// TIA Portal V17 export
// export: Created 2023-04-26T11:43:36.2466218Z, ExportSetting None, DisplayName Totally Integrated Automation Portal, DisplayVersion V17 Update 4, DisplayName TIA Portal Openness, DisplayVersion V17 Update 4, DisplayName TIA Portal Version Control Interface, DisplayVersion V17, DisplayName STEP 7 Professional, DisplayVersion V17 Update 4, DisplayName STEP 7 Safety, DisplayVersion V17, DisplayName WinCC Advanced / Unified PC, DisplayVersion V17 Update 4
FUNCTION "FC_AIn" : Void   // FC14, LAD
TITLE = FC_AIn
{ S7_Optimized_Access := 'FALSE' }
// Analog Input
// stored: SetENOAutomatically false
BEGIN

REGION Network 1: AI 1
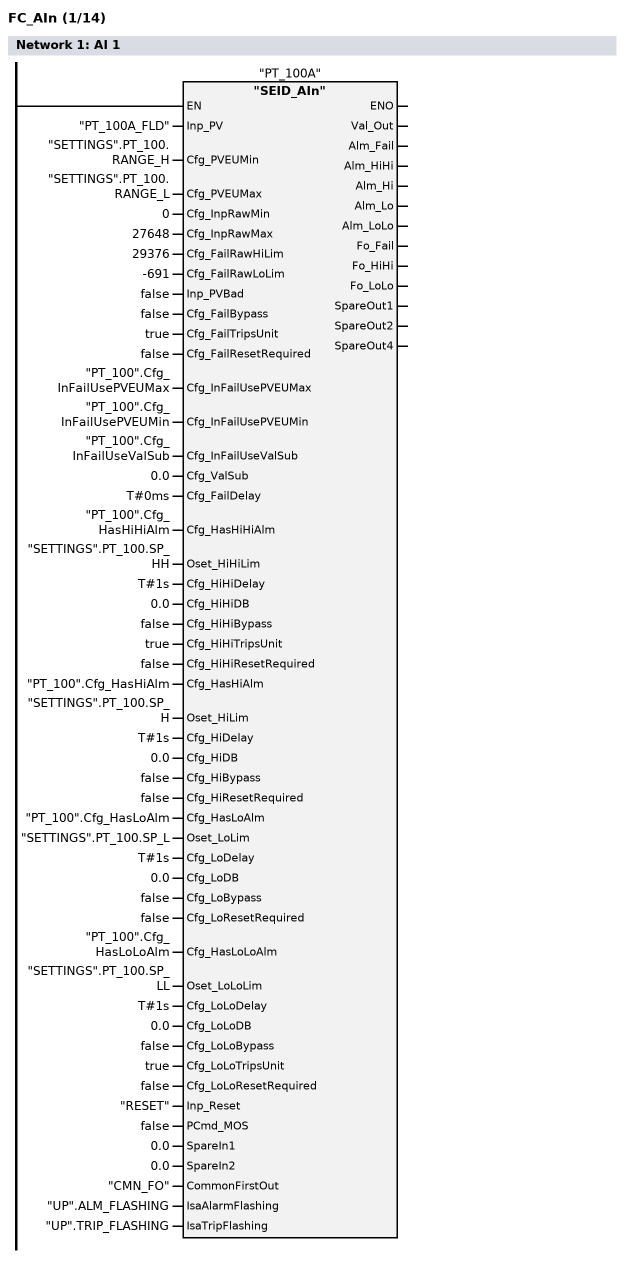
   RUNG wire#powerrail
      "PT_100A"(Inp_PV := "PT_100A_FLD", Cfg_PVEUMin := "SETTINGS".PT_100.RANGE_H, Cfg_PVEUMax := "SETTINGS".PT_100.RANGE_L, Cfg_InpRawMin := 0, Cfg_InpRawMax := 27648, Cfg_FailRawHiLim := 29376, Cfg_FailRawLoLim := -691, Inp_PVBad := false, Cfg_FailBypass := false, Cfg_FailTripsUnit := true, Cfg_FailResetRequired := false, Cfg_InFailUsePVEUMax := "PT_100".Cfg_InFailUsePVEUMax, Cfg_InFailUsePVEUMin := "PT_100".Cfg_InFailUsePVEUMin, Cfg_InFailUseValSub := "PT_100".Cfg_InFailUseValSub, Cfg_ValSub := 0.0, Cfg_FailDelay := T#0ms, Cfg_HasHiHiAlm := "PT_100".Cfg_HasHiHiAlm, Oset_HiHiLim := "SETTINGS".PT_100.SP_HH, Cfg_HiHiDelay := T#1s, Cfg_HiHiDB := 0.0, Cfg_HiHiBypass := false, Cfg_HiHiTripsUnit := true, Cfg_HiHiResetRequired := false, Cfg_HasHiAlm := "PT_100".Cfg_HasHiAlm, Oset_HiLim := "SETTINGS".PT_100.SP_H, Cfg_HiDelay := T#1s, Cfg_HiDB := 0.0, Cfg_HiBypass := false, Cfg_HiResetRequired := false, Cfg_HasLoAlm := "PT_100".Cfg_HasLoAlm, Oset_LoLim := "SETTINGS".PT_100.SP_L, Cfg_LoDelay := T#1s, Cfg_LoDB := 0.0, Cfg_LoBypass := false, Cfg_LoResetRequired := false, Cfg_HasLoLoAlm := "PT_100".Cfg_HasLoLoAlm, Oset_LoLoLim := "SETTINGS".PT_100.SP_LL, Cfg_LoLoDelay := T#1s, Cfg_LoLoDB := 0.0, Cfg_LoLoBypass := false, Cfg_LoLoTripsUnit := true, Cfg_LoLoResetRequired := false, Inp_Reset := "RESET", PCmd_MOS := false, SpareIn1 := 0.0, SpareIn2 := 0.0, CommonFirstOut := "CMN_FO", IsaAlarmFlashing := "UP".ALM_FLASHING, IsaTripFlashing := "UP".TRIP_FLASHING, Val_Out =>, Alm_Fail =>, Alm_HiHi =>, Alm_Hi =>, Alm_Lo =>, Alm_LoLo =>, Fo_Fail =>, Fo_HiHi =>, Fo_LoLo =>, SpareOut1 =>, SpareOut2 =>, SpareOut4 =>)
   END_RUNG
   // the same network as SCL:
   "PT_100A"(Inp_PV := "PT_100A_FLD",   // "SEID_AIn"
             Cfg_PVEUMin := "SETTINGS".PT_100.RANGE_H,
             Cfg_PVEUMax := "SETTINGS".PT_100.RANGE_L,
             Cfg_InpRawMin := 0,
             Cfg_InpRawMax := 27648,
             Cfg_FailRawHiLim := 29376,
             Cfg_FailRawLoLim := -691,
             Inp_PVBad := false,
             Cfg_FailBypass := false,
             Cfg_FailTripsUnit := true,
             Cfg_FailResetRequired := false,
             Cfg_InFailUsePVEUMax := "PT_100".Cfg_InFailUsePVEUMax,
             Cfg_InFailUsePVEUMin := "PT_100".Cfg_InFailUsePVEUMin,
             Cfg_InFailUseValSub := "PT_100".Cfg_InFailUseValSub,
             Cfg_ValSub := 0.0,
             Cfg_FailDelay := T#0ms,
             Cfg_HasHiHiAlm := "PT_100".Cfg_HasHiHiAlm,
             Oset_HiHiLim := "SETTINGS".PT_100.SP_HH,
             Cfg_HiHiDelay := T#1s,
             Cfg_HiHiDB := 0.0,
             Cfg_HiHiBypass := false,
             Cfg_HiHiTripsUnit := true,
             Cfg_HiHiResetRequired := false,
             Cfg_HasHiAlm := "PT_100".Cfg_HasHiAlm,
             Oset_HiLim := "SETTINGS".PT_100.SP_H,
             Cfg_HiDelay := T#1s,
             Cfg_HiDB := 0.0,
             Cfg_HiBypass := false,
             Cfg_HiResetRequired := false,
             Cfg_HasLoAlm := "PT_100".Cfg_HasLoAlm,
             Oset_LoLim := "SETTINGS".PT_100.SP_L,
             Cfg_LoDelay := T#1s,
             Cfg_LoDB := 0.0,
             Cfg_LoBypass := false,
             Cfg_LoResetRequired := false,
             Cfg_HasLoLoAlm := "PT_100".Cfg_HasLoLoAlm,
             Oset_LoLoLim := "SETTINGS".PT_100.SP_LL,
             Cfg_LoLoDelay := T#1s,
             Cfg_LoLoDB := 0.0,
             Cfg_LoLoBypass := false,
             Cfg_LoLoTripsUnit := true,
             Cfg_LoLoResetRequired := false,
             Inp_Reset := "RESET",
             PCmd_MOS := false,
             SpareIn1 := 0.0,
             SpareIn2 := 0.0,
             CommonFirstOut := "CMN_FO",
             IsaAlarmFlashing := "UP".ALM_FLASHING,
             IsaTripFlashing := "UP".TRIP_FLASHING);
END_REGION

REGION Network 2: AI 2
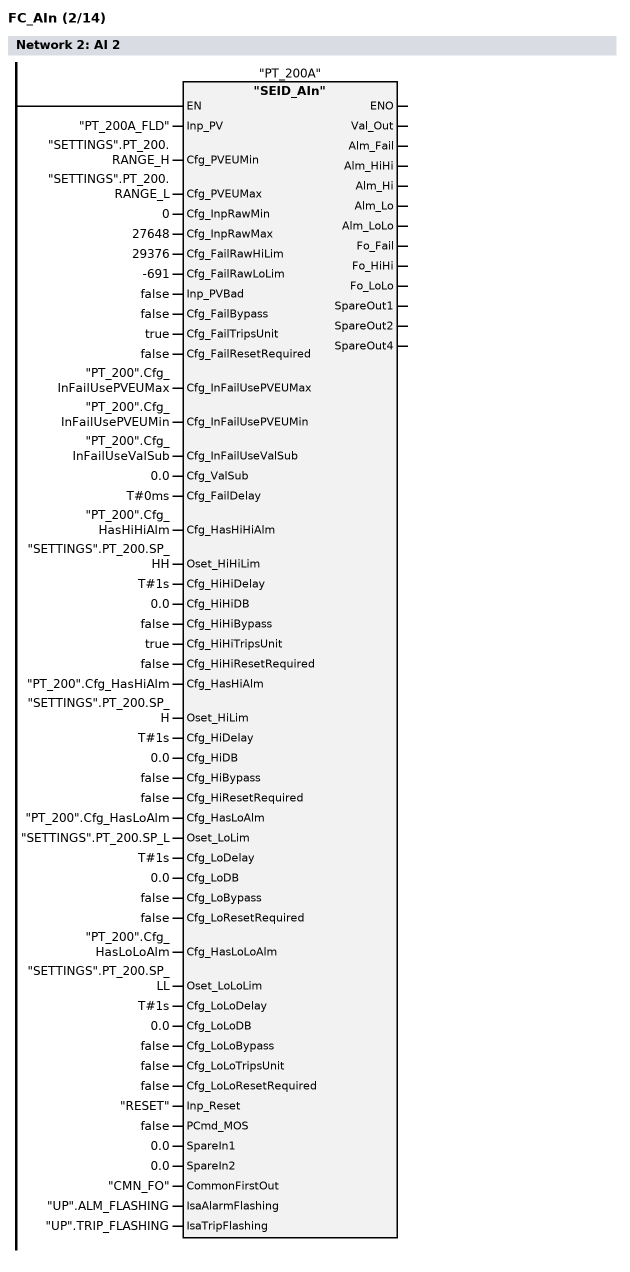
   RUNG wire#powerrail
      "PT_200A"(Inp_PV := "PT_200A_FLD", Cfg_PVEUMin := "SETTINGS".PT_200.RANGE_H, Cfg_PVEUMax := "SETTINGS".PT_200.RANGE_L, Cfg_InpRawMin := 0, Cfg_InpRawMax := 27648, Cfg_FailRawHiLim := 29376, Cfg_FailRawLoLim := -691, Inp_PVBad := false, Cfg_FailBypass := false, Cfg_FailTripsUnit := true, Cfg_FailResetRequired := false, Cfg_InFailUsePVEUMax := "PT_200".Cfg_InFailUsePVEUMax, Cfg_InFailUsePVEUMin := "PT_200".Cfg_InFailUsePVEUMin, Cfg_InFailUseValSub := "PT_200".Cfg_InFailUseValSub, Cfg_ValSub := 0.0, Cfg_FailDelay := T#0ms, Cfg_HasHiHiAlm := "PT_200".Cfg_HasHiHiAlm, Oset_HiHiLim := "SETTINGS".PT_200.SP_HH, Cfg_HiHiDelay := T#1s, Cfg_HiHiDB := 0.0, Cfg_HiHiBypass := false, Cfg_HiHiTripsUnit := true, Cfg_HiHiResetRequired := false, Cfg_HasHiAlm := "PT_200".Cfg_HasHiAlm, Oset_HiLim := "SETTINGS".PT_200.SP_H, Cfg_HiDelay := T#1s, Cfg_HiDB := 0.0, Cfg_HiBypass := false, Cfg_HiResetRequired := false, Cfg_HasLoAlm := "PT_200".Cfg_HasLoAlm, Oset_LoLim := "SETTINGS".PT_200.SP_L, Cfg_LoDelay := T#1s, Cfg_LoDB := 0.0, Cfg_LoBypass := false, Cfg_LoResetRequired := false, Cfg_HasLoLoAlm := "PT_200".Cfg_HasLoLoAlm, Oset_LoLoLim := "SETTINGS".PT_200.SP_LL, Cfg_LoLoDelay := T#1s, Cfg_LoLoDB := 0.0, Cfg_LoLoBypass := false, Cfg_LoLoTripsUnit := false, Cfg_LoLoResetRequired := false, Inp_Reset := "RESET", PCmd_MOS := false, SpareIn1 := 0.0, SpareIn2 := 0.0, CommonFirstOut := "CMN_FO", IsaAlarmFlashing := "UP".ALM_FLASHING, IsaTripFlashing := "UP".TRIP_FLASHING, Val_Out =>, Alm_Fail =>, Alm_HiHi =>, Alm_Hi =>, Alm_Lo =>, Alm_LoLo =>, Fo_Fail =>, Fo_HiHi =>, Fo_LoLo =>, SpareOut1 =>, SpareOut2 =>, SpareOut4 =>)
   END_RUNG
   // the same network as SCL:
   "PT_200A"(Inp_PV := "PT_200A_FLD",   // "SEID_AIn"
             Cfg_PVEUMin := "SETTINGS".PT_200.RANGE_H,
             Cfg_PVEUMax := "SETTINGS".PT_200.RANGE_L,
             Cfg_InpRawMin := 0,
             Cfg_InpRawMax := 27648,
             Cfg_FailRawHiLim := 29376,
             Cfg_FailRawLoLim := -691,
             Inp_PVBad := false,
             Cfg_FailBypass := false,
             Cfg_FailTripsUnit := true,
             Cfg_FailResetRequired := false,
             Cfg_InFailUsePVEUMax := "PT_200".Cfg_InFailUsePVEUMax,
             Cfg_InFailUsePVEUMin := "PT_200".Cfg_InFailUsePVEUMin,
             Cfg_InFailUseValSub := "PT_200".Cfg_InFailUseValSub,
             Cfg_ValSub := 0.0,
             Cfg_FailDelay := T#0ms,
             Cfg_HasHiHiAlm := "PT_200".Cfg_HasHiHiAlm,
             Oset_HiHiLim := "SETTINGS".PT_200.SP_HH,
             Cfg_HiHiDelay := T#1s,
             Cfg_HiHiDB := 0.0,
             Cfg_HiHiBypass := false,
             Cfg_HiHiTripsUnit := true,
             Cfg_HiHiResetRequired := false,
             Cfg_HasHiAlm := "PT_200".Cfg_HasHiAlm,
             Oset_HiLim := "SETTINGS".PT_200.SP_H,
             Cfg_HiDelay := T#1s,
             Cfg_HiDB := 0.0,
             Cfg_HiBypass := false,
             Cfg_HiResetRequired := false,
             Cfg_HasLoAlm := "PT_200".Cfg_HasLoAlm,
             Oset_LoLim := "SETTINGS".PT_200.SP_L,
             Cfg_LoDelay := T#1s,
             Cfg_LoDB := 0.0,
             Cfg_LoBypass := false,
             Cfg_LoResetRequired := false,
             Cfg_HasLoLoAlm := "PT_200".Cfg_HasLoLoAlm,
             Oset_LoLoLim := "SETTINGS".PT_200.SP_LL,
             Cfg_LoLoDelay := T#1s,
             Cfg_LoLoDB := 0.0,
             Cfg_LoLoBypass := false,
             Cfg_LoLoTripsUnit := false,
             Cfg_LoLoResetRequired := false,
             Inp_Reset := "RESET",
             PCmd_MOS := false,
             SpareIn1 := 0.0,
             SpareIn2 := 0.0,
             CommonFirstOut := "CMN_FO",
             IsaAlarmFlashing := "UP".ALM_FLASHING,
             IsaTripFlashing := "UP".TRIP_FLASHING);
END_REGION

REGION Network 3: AI 3
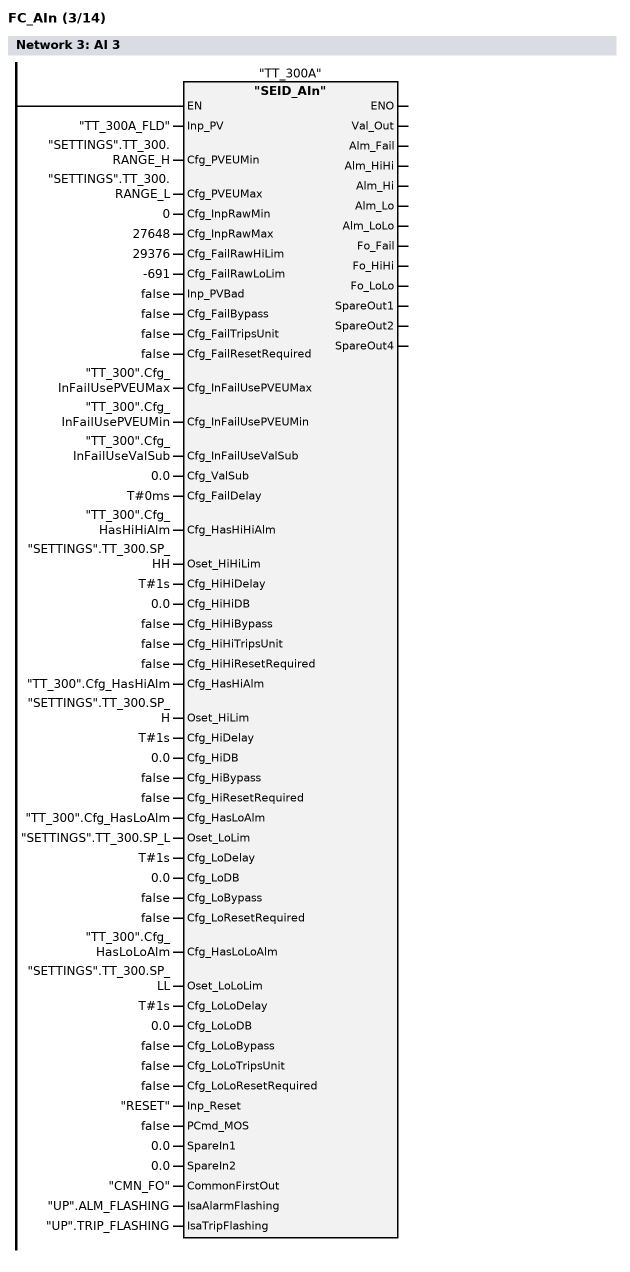
   RUNG wire#powerrail
      "TT_300A"(Inp_PV := "TT_300A_FLD", Cfg_PVEUMin := "SETTINGS".TT_300.RANGE_H, Cfg_PVEUMax := "SETTINGS".TT_300.RANGE_L, Cfg_InpRawMin := 0, Cfg_InpRawMax := 27648, Cfg_FailRawHiLim := 29376, Cfg_FailRawLoLim := -691, Inp_PVBad := false, Cfg_FailBypass := false, Cfg_FailTripsUnit := false, Cfg_FailResetRequired := false, Cfg_InFailUsePVEUMax := "TT_300".Cfg_InFailUsePVEUMax, Cfg_InFailUsePVEUMin := "TT_300".Cfg_InFailUsePVEUMin, Cfg_InFailUseValSub := "TT_300".Cfg_InFailUseValSub, Cfg_ValSub := 0.0, Cfg_FailDelay := T#0ms, Cfg_HasHiHiAlm := "TT_300".Cfg_HasHiHiAlm, Oset_HiHiLim := "SETTINGS".TT_300.SP_HH, Cfg_HiHiDelay := T#1s, Cfg_HiHiDB := 0.0, Cfg_HiHiBypass := false, Cfg_HiHiTripsUnit := false, Cfg_HiHiResetRequired := false, Cfg_HasHiAlm := "TT_300".Cfg_HasHiAlm, Oset_HiLim := "SETTINGS".TT_300.SP_H, Cfg_HiDelay := T#1s, Cfg_HiDB := 0.0, Cfg_HiBypass := false, Cfg_HiResetRequired := false, Cfg_HasLoAlm := "TT_300".Cfg_HasLoAlm, Oset_LoLim := "SETTINGS".TT_300.SP_L, Cfg_LoDelay := T#1s, Cfg_LoDB := 0.0, Cfg_LoBypass := false, Cfg_LoResetRequired := false, Cfg_HasLoLoAlm := "TT_300".Cfg_HasLoLoAlm, Oset_LoLoLim := "SETTINGS".TT_300.SP_LL, Cfg_LoLoDelay := T#1s, Cfg_LoLoDB := 0.0, Cfg_LoLoBypass := false, Cfg_LoLoTripsUnit := false, Cfg_LoLoResetRequired := false, Inp_Reset := "RESET", PCmd_MOS := false, SpareIn1 := 0.0, SpareIn2 := 0.0, CommonFirstOut := "CMN_FO", IsaAlarmFlashing := "UP".ALM_FLASHING, IsaTripFlashing := "UP".TRIP_FLASHING, Val_Out =>, Alm_Fail =>, Alm_HiHi =>, Alm_Hi =>, Alm_Lo =>, Alm_LoLo =>, Fo_Fail =>, Fo_HiHi =>, Fo_LoLo =>, SpareOut1 =>, SpareOut2 =>, SpareOut4 =>)
   END_RUNG
   // the same network as SCL:
   "TT_300A"(Inp_PV := "TT_300A_FLD",   // "SEID_AIn"
             Cfg_PVEUMin := "SETTINGS".TT_300.RANGE_H,
             Cfg_PVEUMax := "SETTINGS".TT_300.RANGE_L,
             Cfg_InpRawMin := 0,
             Cfg_InpRawMax := 27648,
             Cfg_FailRawHiLim := 29376,
             Cfg_FailRawLoLim := -691,
             Inp_PVBad := false,
             Cfg_FailBypass := false,
             Cfg_FailTripsUnit := false,
             Cfg_FailResetRequired := false,
             Cfg_InFailUsePVEUMax := "TT_300".Cfg_InFailUsePVEUMax,
             Cfg_InFailUsePVEUMin := "TT_300".Cfg_InFailUsePVEUMin,
             Cfg_InFailUseValSub := "TT_300".Cfg_InFailUseValSub,
             Cfg_ValSub := 0.0,
             Cfg_FailDelay := T#0ms,
             Cfg_HasHiHiAlm := "TT_300".Cfg_HasHiHiAlm,
             Oset_HiHiLim := "SETTINGS".TT_300.SP_HH,
             Cfg_HiHiDelay := T#1s,
             Cfg_HiHiDB := 0.0,
             Cfg_HiHiBypass := false,
             Cfg_HiHiTripsUnit := false,
             Cfg_HiHiResetRequired := false,
             Cfg_HasHiAlm := "TT_300".Cfg_HasHiAlm,
             Oset_HiLim := "SETTINGS".TT_300.SP_H,
             Cfg_HiDelay := T#1s,
             Cfg_HiDB := 0.0,
             Cfg_HiBypass := false,
             Cfg_HiResetRequired := false,
             Cfg_HasLoAlm := "TT_300".Cfg_HasLoAlm,
             Oset_LoLim := "SETTINGS".TT_300.SP_L,
             Cfg_LoDelay := T#1s,
             Cfg_LoDB := 0.0,
             Cfg_LoBypass := false,
             Cfg_LoResetRequired := false,
             Cfg_HasLoLoAlm := "TT_300".Cfg_HasLoLoAlm,
             Oset_LoLoLim := "SETTINGS".TT_300.SP_LL,
             Cfg_LoLoDelay := T#1s,
             Cfg_LoLoDB := 0.0,
             Cfg_LoLoBypass := false,
             Cfg_LoLoTripsUnit := false,
             Cfg_LoLoResetRequired := false,
             Inp_Reset := "RESET",
             PCmd_MOS := false,
             SpareIn1 := 0.0,
             SpareIn2 := 0.0,
             CommonFirstOut := "CMN_FO",
             IsaAlarmFlashing := "UP".ALM_FLASHING,
             IsaTripFlashing := "UP".TRIP_FLASHING);
END_REGION

REGION Network 4: AI 4
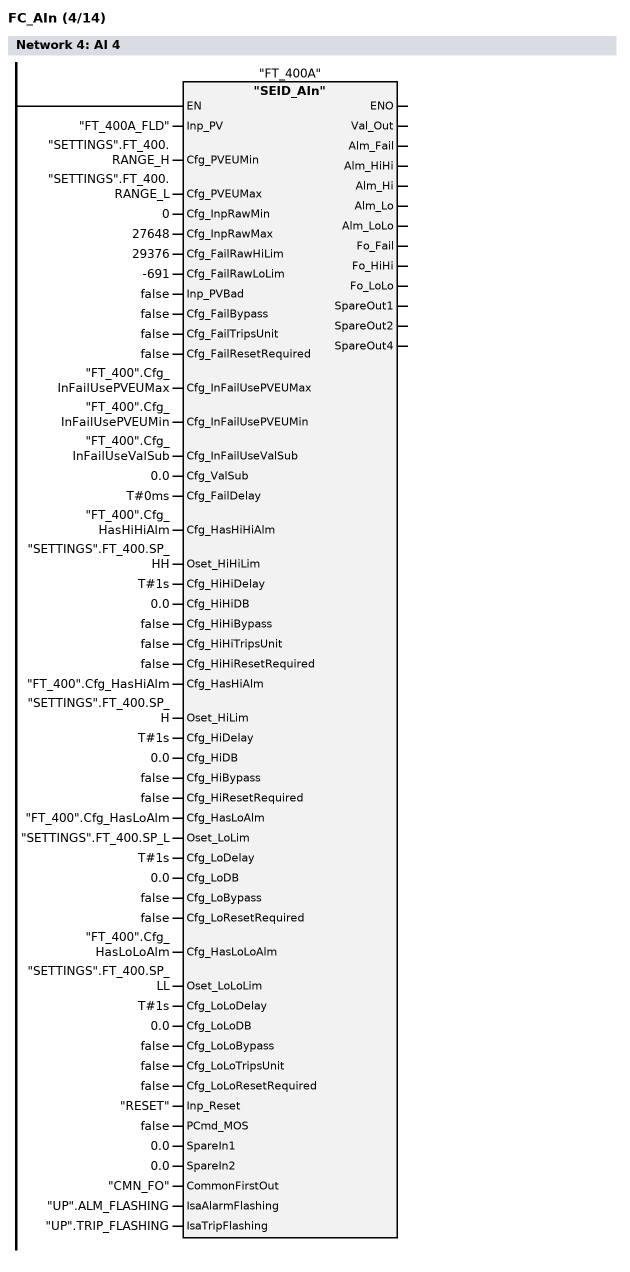
   RUNG wire#powerrail
      "FT_400A"(Inp_PV := "FT_400A_FLD", Cfg_PVEUMin := "SETTINGS".FT_400.RANGE_H, Cfg_PVEUMax := "SETTINGS".FT_400.RANGE_L, Cfg_InpRawMin := 0, Cfg_InpRawMax := 27648, Cfg_FailRawHiLim := 29376, Cfg_FailRawLoLim := -691, Inp_PVBad := false, Cfg_FailBypass := false, Cfg_FailTripsUnit := false, Cfg_FailResetRequired := false, Cfg_InFailUsePVEUMax := "FT_400".Cfg_InFailUsePVEUMax, Cfg_InFailUsePVEUMin := "FT_400".Cfg_InFailUsePVEUMin, Cfg_InFailUseValSub := "FT_400".Cfg_InFailUseValSub, Cfg_ValSub := 0.0, Cfg_FailDelay := T#0ms, Cfg_HasHiHiAlm := "FT_400".Cfg_HasHiHiAlm, Oset_HiHiLim := "SETTINGS".FT_400.SP_HH, Cfg_HiHiDelay := T#1s, Cfg_HiHiDB := 0.0, Cfg_HiHiBypass := false, Cfg_HiHiTripsUnit := false, Cfg_HiHiResetRequired := false, Cfg_HasHiAlm := "FT_400".Cfg_HasHiAlm, Oset_HiLim := "SETTINGS".FT_400.SP_H, Cfg_HiDelay := T#1s, Cfg_HiDB := 0.0, Cfg_HiBypass := false, Cfg_HiResetRequired := false, Cfg_HasLoAlm := "FT_400".Cfg_HasLoAlm, Oset_LoLim := "SETTINGS".FT_400.SP_L, Cfg_LoDelay := T#1s, Cfg_LoDB := 0.0, Cfg_LoBypass := false, Cfg_LoResetRequired := false, Cfg_HasLoLoAlm := "FT_400".Cfg_HasLoLoAlm, Oset_LoLoLim := "SETTINGS".FT_400.SP_LL, Cfg_LoLoDelay := T#1s, Cfg_LoLoDB := 0.0, Cfg_LoLoBypass := false, Cfg_LoLoTripsUnit := false, Cfg_LoLoResetRequired := false, Inp_Reset := "RESET", PCmd_MOS := false, SpareIn1 := 0.0, SpareIn2 := 0.0, CommonFirstOut := "CMN_FO", IsaAlarmFlashing := "UP".ALM_FLASHING, IsaTripFlashing := "UP".TRIP_FLASHING, Val_Out =>, Alm_Fail =>, Alm_HiHi =>, Alm_Hi =>, Alm_Lo =>, Alm_LoLo =>, Fo_Fail =>, Fo_HiHi =>, Fo_LoLo =>, SpareOut1 =>, SpareOut2 =>, SpareOut4 =>)
   END_RUNG
   // the same network as SCL:
   "FT_400A"(Inp_PV := "FT_400A_FLD",   // "SEID_AIn"
             Cfg_PVEUMin := "SETTINGS".FT_400.RANGE_H,
             Cfg_PVEUMax := "SETTINGS".FT_400.RANGE_L,
             Cfg_InpRawMin := 0,
             Cfg_InpRawMax := 27648,
             Cfg_FailRawHiLim := 29376,
             Cfg_FailRawLoLim := -691,
             Inp_PVBad := false,
             Cfg_FailBypass := false,
             Cfg_FailTripsUnit := false,
             Cfg_FailResetRequired := false,
             Cfg_InFailUsePVEUMax := "FT_400".Cfg_InFailUsePVEUMax,
             Cfg_InFailUsePVEUMin := "FT_400".Cfg_InFailUsePVEUMin,
             Cfg_InFailUseValSub := "FT_400".Cfg_InFailUseValSub,
             Cfg_ValSub := 0.0,
             Cfg_FailDelay := T#0ms,
             Cfg_HasHiHiAlm := "FT_400".Cfg_HasHiHiAlm,
             Oset_HiHiLim := "SETTINGS".FT_400.SP_HH,
             Cfg_HiHiDelay := T#1s,
             Cfg_HiHiDB := 0.0,
             Cfg_HiHiBypass := false,
             Cfg_HiHiTripsUnit := false,
             Cfg_HiHiResetRequired := false,
             Cfg_HasHiAlm := "FT_400".Cfg_HasHiAlm,
             Oset_HiLim := "SETTINGS".FT_400.SP_H,
             Cfg_HiDelay := T#1s,
             Cfg_HiDB := 0.0,
             Cfg_HiBypass := false,
             Cfg_HiResetRequired := false,
             Cfg_HasLoAlm := "FT_400".Cfg_HasLoAlm,
             Oset_LoLim := "SETTINGS".FT_400.SP_L,
             Cfg_LoDelay := T#1s,
             Cfg_LoDB := 0.0,
             Cfg_LoBypass := false,
             Cfg_LoResetRequired := false,
             Cfg_HasLoLoAlm := "FT_400".Cfg_HasLoLoAlm,
             Oset_LoLoLim := "SETTINGS".FT_400.SP_LL,
             Cfg_LoLoDelay := T#1s,
             Cfg_LoLoDB := 0.0,
             Cfg_LoLoBypass := false,
             Cfg_LoLoTripsUnit := false,
             Cfg_LoLoResetRequired := false,
             Inp_Reset := "RESET",
             PCmd_MOS := false,
             SpareIn1 := 0.0,
             SpareIn2 := 0.0,
             CommonFirstOut := "CMN_FO",
             IsaAlarmFlashing := "UP".ALM_FLASHING,
             IsaTripFlashing := "UP".TRIP_FLASHING);
END_REGION

REGION Network 5: AI 5
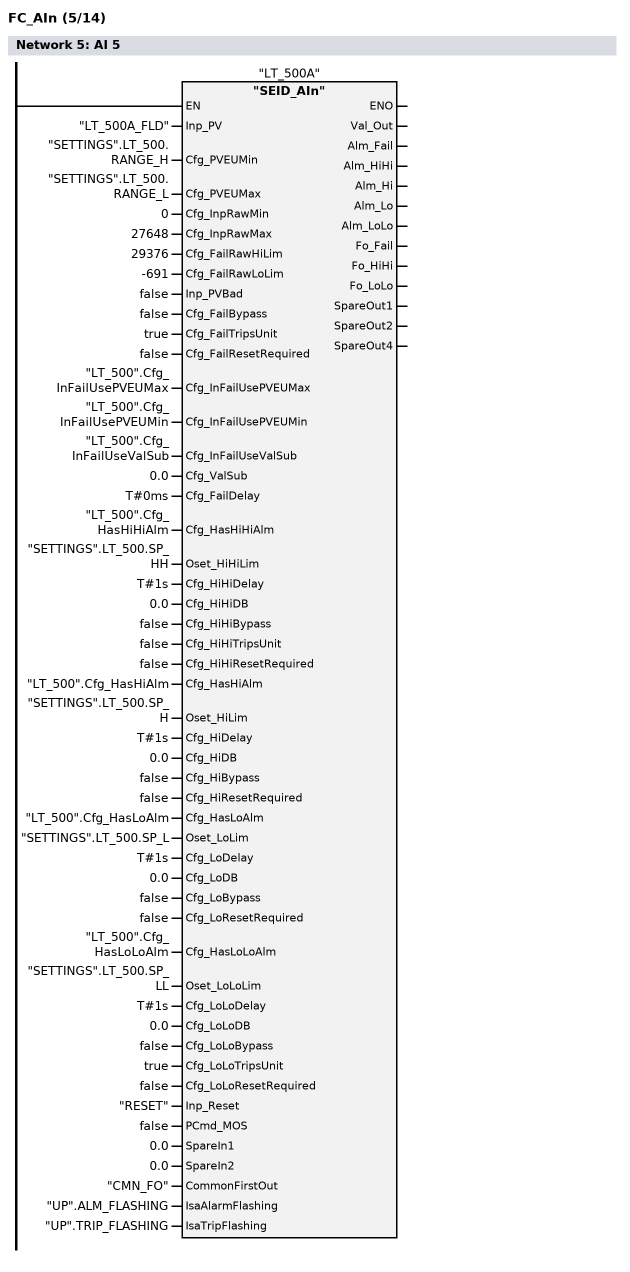
   RUNG wire#powerrail
      "LT_500A"(Inp_PV := "LT_500A_FLD", Cfg_PVEUMin := "SETTINGS".LT_500.RANGE_H, Cfg_PVEUMax := "SETTINGS".LT_500.RANGE_L, Cfg_InpRawMin := 0, Cfg_InpRawMax := 27648, Cfg_FailRawHiLim := 29376, Cfg_FailRawLoLim := -691, Inp_PVBad := false, Cfg_FailBypass := false, Cfg_FailTripsUnit := true, Cfg_FailResetRequired := false, Cfg_InFailUsePVEUMax := "LT_500".Cfg_InFailUsePVEUMax, Cfg_InFailUsePVEUMin := "LT_500".Cfg_InFailUsePVEUMin, Cfg_InFailUseValSub := "LT_500".Cfg_InFailUseValSub, Cfg_ValSub := 0.0, Cfg_FailDelay := T#0ms, Cfg_HasHiHiAlm := "LT_500".Cfg_HasHiHiAlm, Oset_HiHiLim := "SETTINGS".LT_500.SP_HH, Cfg_HiHiDelay := T#1s, Cfg_HiHiDB := 0.0, Cfg_HiHiBypass := false, Cfg_HiHiTripsUnit := false, Cfg_HiHiResetRequired := false, Cfg_HasHiAlm := "LT_500".Cfg_HasHiAlm, Oset_HiLim := "SETTINGS".LT_500.SP_H, Cfg_HiDelay := T#1s, Cfg_HiDB := 0.0, Cfg_HiBypass := false, Cfg_HiResetRequired := false, Cfg_HasLoAlm := "LT_500".Cfg_HasLoAlm, Oset_LoLim := "SETTINGS".LT_500.SP_L, Cfg_LoDelay := T#1s, Cfg_LoDB := 0.0, Cfg_LoBypass := false, Cfg_LoResetRequired := false, Cfg_HasLoLoAlm := "LT_500".Cfg_HasLoLoAlm, Oset_LoLoLim := "SETTINGS".LT_500.SP_LL, Cfg_LoLoDelay := T#1s, Cfg_LoLoDB := 0.0, Cfg_LoLoBypass := false, Cfg_LoLoTripsUnit := true, Cfg_LoLoResetRequired := false, Inp_Reset := "RESET", PCmd_MOS := false, SpareIn1 := 0.0, SpareIn2 := 0.0, CommonFirstOut := "CMN_FO", IsaAlarmFlashing := "UP".ALM_FLASHING, IsaTripFlashing := "UP".TRIP_FLASHING, Val_Out =>, Alm_Fail =>, Alm_HiHi =>, Alm_Hi =>, Alm_Lo =>, Alm_LoLo =>, Fo_Fail =>, Fo_HiHi =>, Fo_LoLo =>, SpareOut1 =>, SpareOut2 =>, SpareOut4 =>)
   END_RUNG
   // the same network as SCL:
   "LT_500A"(Inp_PV := "LT_500A_FLD",   // "SEID_AIn"
             Cfg_PVEUMin := "SETTINGS".LT_500.RANGE_H,
             Cfg_PVEUMax := "SETTINGS".LT_500.RANGE_L,
             Cfg_InpRawMin := 0,
             Cfg_InpRawMax := 27648,
             Cfg_FailRawHiLim := 29376,
             Cfg_FailRawLoLim := -691,
             Inp_PVBad := false,
             Cfg_FailBypass := false,
             Cfg_FailTripsUnit := true,
             Cfg_FailResetRequired := false,
             Cfg_InFailUsePVEUMax := "LT_500".Cfg_InFailUsePVEUMax,
             Cfg_InFailUsePVEUMin := "LT_500".Cfg_InFailUsePVEUMin,
             Cfg_InFailUseValSub := "LT_500".Cfg_InFailUseValSub,
             Cfg_ValSub := 0.0,
             Cfg_FailDelay := T#0ms,
             Cfg_HasHiHiAlm := "LT_500".Cfg_HasHiHiAlm,
             Oset_HiHiLim := "SETTINGS".LT_500.SP_HH,
             Cfg_HiHiDelay := T#1s,
             Cfg_HiHiDB := 0.0,
             Cfg_HiHiBypass := false,
             Cfg_HiHiTripsUnit := false,
             Cfg_HiHiResetRequired := false,
             Cfg_HasHiAlm := "LT_500".Cfg_HasHiAlm,
             Oset_HiLim := "SETTINGS".LT_500.SP_H,
             Cfg_HiDelay := T#1s,
             Cfg_HiDB := 0.0,
             Cfg_HiBypass := false,
             Cfg_HiResetRequired := false,
             Cfg_HasLoAlm := "LT_500".Cfg_HasLoAlm,
             Oset_LoLim := "SETTINGS".LT_500.SP_L,
             Cfg_LoDelay := T#1s,
             Cfg_LoDB := 0.0,
             Cfg_LoBypass := false,
             Cfg_LoResetRequired := false,
             Cfg_HasLoLoAlm := "LT_500".Cfg_HasLoLoAlm,
             Oset_LoLoLim := "SETTINGS".LT_500.SP_LL,
             Cfg_LoLoDelay := T#1s,
             Cfg_LoLoDB := 0.0,
             Cfg_LoLoBypass := false,
             Cfg_LoLoTripsUnit := true,
             Cfg_LoLoResetRequired := false,
             Inp_Reset := "RESET",
             PCmd_MOS := false,
             SpareIn1 := 0.0,
             SpareIn2 := 0.0,
             CommonFirstOut := "CMN_FO",
             IsaAlarmFlashing := "UP".ALM_FLASHING,
             IsaTripFlashing := "UP".TRIP_FLASHING);
END_REGION

REGION Network 6: AI 6
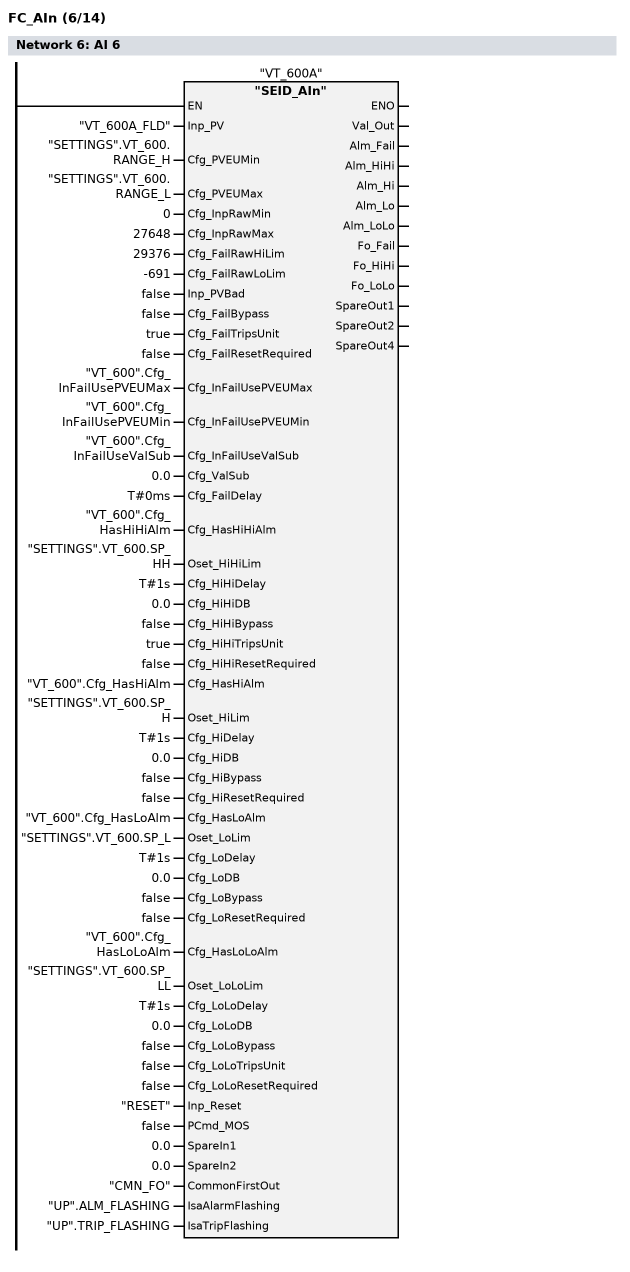
   RUNG wire#powerrail
      "VT_600A"(Inp_PV := "VT_600A_FLD", Cfg_PVEUMin := "SETTINGS".VT_600.RANGE_H, Cfg_PVEUMax := "SETTINGS".VT_600.RANGE_L, Cfg_InpRawMin := 0, Cfg_InpRawMax := 27648, Cfg_FailRawHiLim := 29376, Cfg_FailRawLoLim := -691, Inp_PVBad := false, Cfg_FailBypass := false, Cfg_FailTripsUnit := true, Cfg_FailResetRequired := false, Cfg_InFailUsePVEUMax := "VT_600".Cfg_InFailUsePVEUMax, Cfg_InFailUsePVEUMin := "VT_600".Cfg_InFailUsePVEUMin, Cfg_InFailUseValSub := "VT_600".Cfg_InFailUseValSub, Cfg_ValSub := 0.0, Cfg_FailDelay := T#0ms, Cfg_HasHiHiAlm := "VT_600".Cfg_HasHiHiAlm, Oset_HiHiLim := "SETTINGS".VT_600.SP_HH, Cfg_HiHiDelay := T#1s, Cfg_HiHiDB := 0.0, Cfg_HiHiBypass := false, Cfg_HiHiTripsUnit := true, Cfg_HiHiResetRequired := false, Cfg_HasHiAlm := "VT_600".Cfg_HasHiAlm, Oset_HiLim := "SETTINGS".VT_600.SP_H, Cfg_HiDelay := T#1s, Cfg_HiDB := 0.0, Cfg_HiBypass := false, Cfg_HiResetRequired := false, Cfg_HasLoAlm := "VT_600".Cfg_HasLoAlm, Oset_LoLim := "SETTINGS".VT_600.SP_L, Cfg_LoDelay := T#1s, Cfg_LoDB := 0.0, Cfg_LoBypass := false, Cfg_LoResetRequired := false, Cfg_HasLoLoAlm := "VT_600".Cfg_HasLoLoAlm, Oset_LoLoLim := "SETTINGS".VT_600.SP_LL, Cfg_LoLoDelay := T#1s, Cfg_LoLoDB := 0.0, Cfg_LoLoBypass := false, Cfg_LoLoTripsUnit := false, Cfg_LoLoResetRequired := false, Inp_Reset := "RESET", PCmd_MOS := false, SpareIn1 := 0.0, SpareIn2 := 0.0, CommonFirstOut := "CMN_FO", IsaAlarmFlashing := "UP".ALM_FLASHING, IsaTripFlashing := "UP".TRIP_FLASHING, Val_Out =>, Alm_Fail =>, Alm_HiHi =>, Alm_Hi =>, Alm_Lo =>, Alm_LoLo =>, Fo_Fail =>, Fo_HiHi =>, Fo_LoLo =>, SpareOut1 =>, SpareOut2 =>, SpareOut4 =>)
   END_RUNG
   // the same network as SCL:
   "VT_600A"(Inp_PV := "VT_600A_FLD",   // "SEID_AIn"
             Cfg_PVEUMin := "SETTINGS".VT_600.RANGE_H,
             Cfg_PVEUMax := "SETTINGS".VT_600.RANGE_L,
             Cfg_InpRawMin := 0,
             Cfg_InpRawMax := 27648,
             Cfg_FailRawHiLim := 29376,
             Cfg_FailRawLoLim := -691,
             Inp_PVBad := false,
             Cfg_FailBypass := false,
             Cfg_FailTripsUnit := true,
             Cfg_FailResetRequired := false,
             Cfg_InFailUsePVEUMax := "VT_600".Cfg_InFailUsePVEUMax,
             Cfg_InFailUsePVEUMin := "VT_600".Cfg_InFailUsePVEUMin,
             Cfg_InFailUseValSub := "VT_600".Cfg_InFailUseValSub,
             Cfg_ValSub := 0.0,
             Cfg_FailDelay := T#0ms,
             Cfg_HasHiHiAlm := "VT_600".Cfg_HasHiHiAlm,
             Oset_HiHiLim := "SETTINGS".VT_600.SP_HH,
             Cfg_HiHiDelay := T#1s,
             Cfg_HiHiDB := 0.0,
             Cfg_HiHiBypass := false,
             Cfg_HiHiTripsUnit := true,
             Cfg_HiHiResetRequired := false,
             Cfg_HasHiAlm := "VT_600".Cfg_HasHiAlm,
             Oset_HiLim := "SETTINGS".VT_600.SP_H,
             Cfg_HiDelay := T#1s,
             Cfg_HiDB := 0.0,
             Cfg_HiBypass := false,
             Cfg_HiResetRequired := false,
             Cfg_HasLoAlm := "VT_600".Cfg_HasLoAlm,
             Oset_LoLim := "SETTINGS".VT_600.SP_L,
             Cfg_LoDelay := T#1s,
             Cfg_LoDB := 0.0,
             Cfg_LoBypass := false,
             Cfg_LoResetRequired := false,
             Cfg_HasLoLoAlm := "VT_600".Cfg_HasLoLoAlm,
             Oset_LoLoLim := "SETTINGS".VT_600.SP_LL,
             Cfg_LoLoDelay := T#1s,
             Cfg_LoLoDB := 0.0,
             Cfg_LoLoBypass := false,
             Cfg_LoLoTripsUnit := false,
             Cfg_LoLoResetRequired := false,
             Inp_Reset := "RESET",
             PCmd_MOS := false,
             SpareIn1 := 0.0,
             SpareIn2 := 0.0,
             CommonFirstOut := "CMN_FO",
             IsaAlarmFlashing := "UP".ALM_FLASHING,
             IsaTripFlashing := "UP".TRIP_FLASHING);
END_REGION

REGION Network 7: AI 7
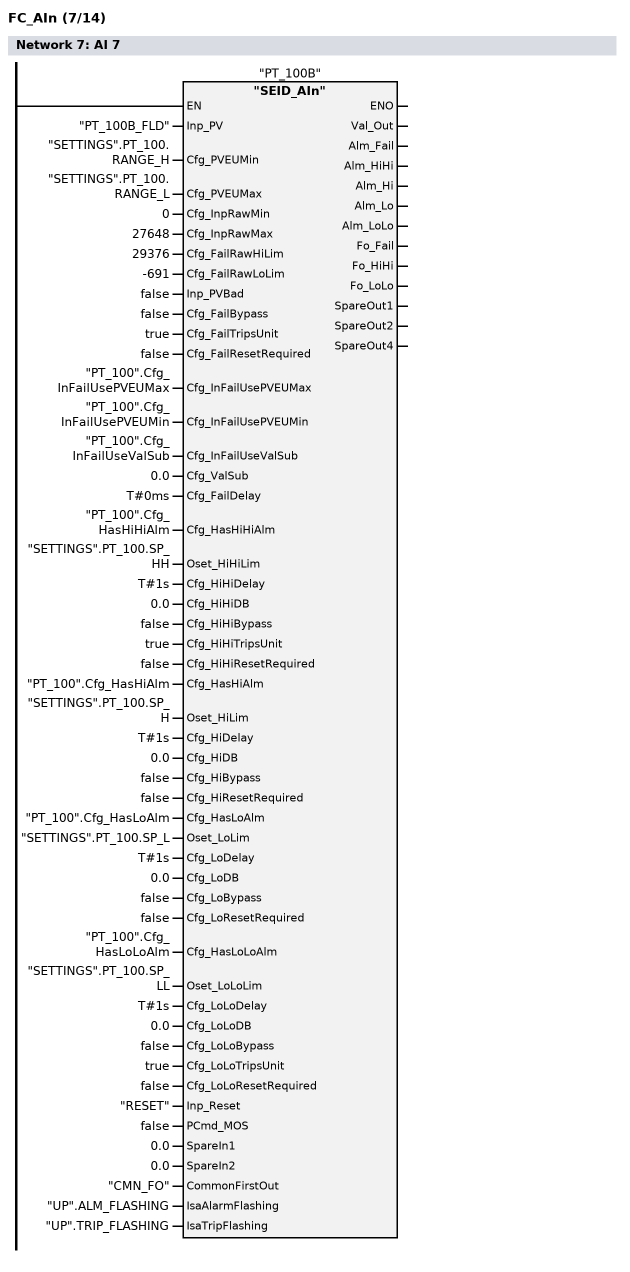
   RUNG wire#powerrail
      "PT_100B"(Inp_PV := "PT_100B_FLD", Cfg_PVEUMin := "SETTINGS".PT_100.RANGE_H, Cfg_PVEUMax := "SETTINGS".PT_100.RANGE_L, Cfg_InpRawMin := 0, Cfg_InpRawMax := 27648, Cfg_FailRawHiLim := 29376, Cfg_FailRawLoLim := -691, Inp_PVBad := false, Cfg_FailBypass := false, Cfg_FailTripsUnit := true, Cfg_FailResetRequired := false, Cfg_InFailUsePVEUMax := "PT_100".Cfg_InFailUsePVEUMax, Cfg_InFailUsePVEUMin := "PT_100".Cfg_InFailUsePVEUMin, Cfg_InFailUseValSub := "PT_100".Cfg_InFailUseValSub, Cfg_ValSub := 0.0, Cfg_FailDelay := T#0ms, Cfg_HasHiHiAlm := "PT_100".Cfg_HasHiHiAlm, Oset_HiHiLim := "SETTINGS".PT_100.SP_HH, Cfg_HiHiDelay := T#1s, Cfg_HiHiDB := 0.0, Cfg_HiHiBypass := false, Cfg_HiHiTripsUnit := true, Cfg_HiHiResetRequired := false, Cfg_HasHiAlm := "PT_100".Cfg_HasHiAlm, Oset_HiLim := "SETTINGS".PT_100.SP_H, Cfg_HiDelay := T#1s, Cfg_HiDB := 0.0, Cfg_HiBypass := false, Cfg_HiResetRequired := false, Cfg_HasLoAlm := "PT_100".Cfg_HasLoAlm, Oset_LoLim := "SETTINGS".PT_100.SP_L, Cfg_LoDelay := T#1s, Cfg_LoDB := 0.0, Cfg_LoBypass := false, Cfg_LoResetRequired := false, Cfg_HasLoLoAlm := "PT_100".Cfg_HasLoLoAlm, Oset_LoLoLim := "SETTINGS".PT_100.SP_LL, Cfg_LoLoDelay := T#1s, Cfg_LoLoDB := 0.0, Cfg_LoLoBypass := false, Cfg_LoLoTripsUnit := true, Cfg_LoLoResetRequired := false, Inp_Reset := "RESET", PCmd_MOS := false, SpareIn1 := 0.0, SpareIn2 := 0.0, CommonFirstOut := "CMN_FO", IsaAlarmFlashing := "UP".ALM_FLASHING, IsaTripFlashing := "UP".TRIP_FLASHING, Val_Out =>, Alm_Fail =>, Alm_HiHi =>, Alm_Hi =>, Alm_Lo =>, Alm_LoLo =>, Fo_Fail =>, Fo_HiHi =>, Fo_LoLo =>, SpareOut1 =>, SpareOut2 =>, SpareOut4 =>)
   END_RUNG
   // the same network as SCL:
   "PT_100B"(Inp_PV := "PT_100B_FLD",   // "SEID_AIn"
             Cfg_PVEUMin := "SETTINGS".PT_100.RANGE_H,
             Cfg_PVEUMax := "SETTINGS".PT_100.RANGE_L,
             Cfg_InpRawMin := 0,
             Cfg_InpRawMax := 27648,
             Cfg_FailRawHiLim := 29376,
             Cfg_FailRawLoLim := -691,
             Inp_PVBad := false,
             Cfg_FailBypass := false,
             Cfg_FailTripsUnit := true,
             Cfg_FailResetRequired := false,
             Cfg_InFailUsePVEUMax := "PT_100".Cfg_InFailUsePVEUMax,
             Cfg_InFailUsePVEUMin := "PT_100".Cfg_InFailUsePVEUMin,
             Cfg_InFailUseValSub := "PT_100".Cfg_InFailUseValSub,
             Cfg_ValSub := 0.0,
             Cfg_FailDelay := T#0ms,
             Cfg_HasHiHiAlm := "PT_100".Cfg_HasHiHiAlm,
             Oset_HiHiLim := "SETTINGS".PT_100.SP_HH,
             Cfg_HiHiDelay := T#1s,
             Cfg_HiHiDB := 0.0,
             Cfg_HiHiBypass := false,
             Cfg_HiHiTripsUnit := true,
             Cfg_HiHiResetRequired := false,
             Cfg_HasHiAlm := "PT_100".Cfg_HasHiAlm,
             Oset_HiLim := "SETTINGS".PT_100.SP_H,
             Cfg_HiDelay := T#1s,
             Cfg_HiDB := 0.0,
             Cfg_HiBypass := false,
             Cfg_HiResetRequired := false,
             Cfg_HasLoAlm := "PT_100".Cfg_HasLoAlm,
             Oset_LoLim := "SETTINGS".PT_100.SP_L,
             Cfg_LoDelay := T#1s,
             Cfg_LoDB := 0.0,
             Cfg_LoBypass := false,
             Cfg_LoResetRequired := false,
             Cfg_HasLoLoAlm := "PT_100".Cfg_HasLoLoAlm,
             Oset_LoLoLim := "SETTINGS".PT_100.SP_LL,
             Cfg_LoLoDelay := T#1s,
             Cfg_LoLoDB := 0.0,
             Cfg_LoLoBypass := false,
             Cfg_LoLoTripsUnit := true,
             Cfg_LoLoResetRequired := false,
             Inp_Reset := "RESET",
             PCmd_MOS := false,
             SpareIn1 := 0.0,
             SpareIn2 := 0.0,
             CommonFirstOut := "CMN_FO",
             IsaAlarmFlashing := "UP".ALM_FLASHING,
             IsaTripFlashing := "UP".TRIP_FLASHING);
END_REGION

REGION Network 8: AI 8
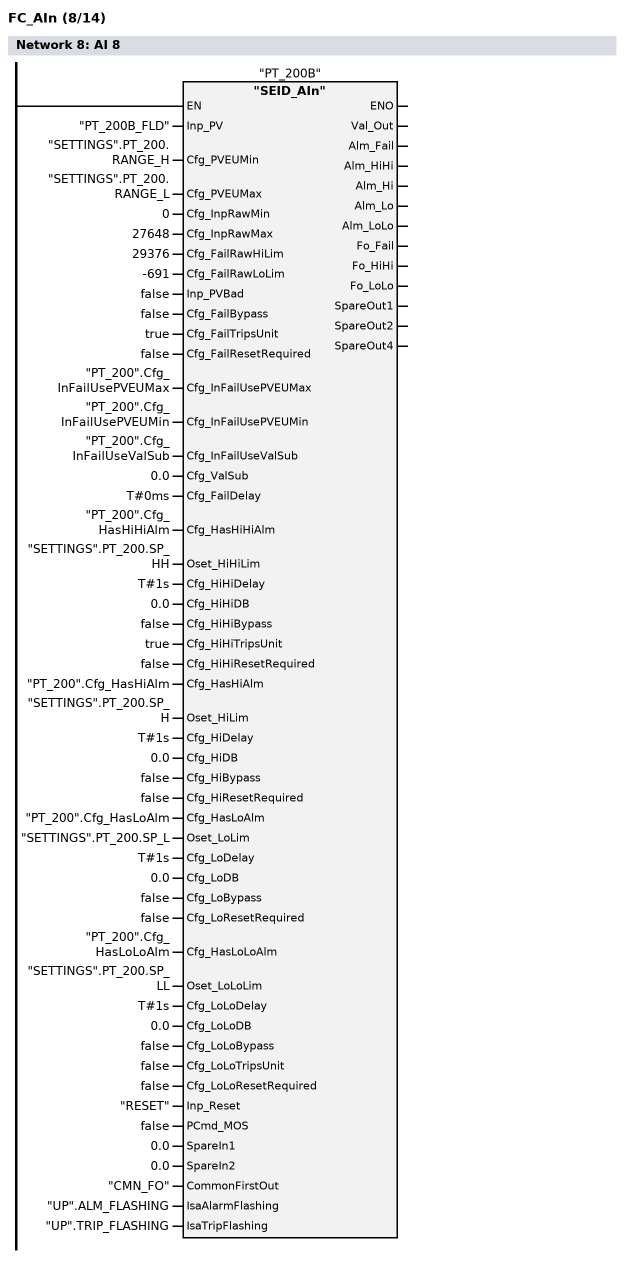
   RUNG wire#powerrail
      "PT_200B"(Inp_PV := "PT_200B_FLD", Cfg_PVEUMin := "SETTINGS".PT_200.RANGE_H, Cfg_PVEUMax := "SETTINGS".PT_200.RANGE_L, Cfg_InpRawMin := 0, Cfg_InpRawMax := 27648, Cfg_FailRawHiLim := 29376, Cfg_FailRawLoLim := -691, Inp_PVBad := false, Cfg_FailBypass := false, Cfg_FailTripsUnit := true, Cfg_FailResetRequired := false, Cfg_InFailUsePVEUMax := "PT_200".Cfg_InFailUsePVEUMax, Cfg_InFailUsePVEUMin := "PT_200".Cfg_InFailUsePVEUMin, Cfg_InFailUseValSub := "PT_200".Cfg_InFailUseValSub, Cfg_ValSub := 0.0, Cfg_FailDelay := T#0ms, Cfg_HasHiHiAlm := "PT_200".Cfg_HasHiHiAlm, Oset_HiHiLim := "SETTINGS".PT_200.SP_HH, Cfg_HiHiDelay := T#1s, Cfg_HiHiDB := 0.0, Cfg_HiHiBypass := false, Cfg_HiHiTripsUnit := true, Cfg_HiHiResetRequired := false, Cfg_HasHiAlm := "PT_200".Cfg_HasHiAlm, Oset_HiLim := "SETTINGS".PT_200.SP_H, Cfg_HiDelay := T#1s, Cfg_HiDB := 0.0, Cfg_HiBypass := false, Cfg_HiResetRequired := false, Cfg_HasLoAlm := "PT_200".Cfg_HasLoAlm, Oset_LoLim := "SETTINGS".PT_200.SP_L, Cfg_LoDelay := T#1s, Cfg_LoDB := 0.0, Cfg_LoBypass := false, Cfg_LoResetRequired := false, Cfg_HasLoLoAlm := "PT_200".Cfg_HasLoLoAlm, Oset_LoLoLim := "SETTINGS".PT_200.SP_LL, Cfg_LoLoDelay := T#1s, Cfg_LoLoDB := 0.0, Cfg_LoLoBypass := false, Cfg_LoLoTripsUnit := false, Cfg_LoLoResetRequired := false, Inp_Reset := "RESET", PCmd_MOS := false, SpareIn1 := 0.0, SpareIn2 := 0.0, CommonFirstOut := "CMN_FO", IsaAlarmFlashing := "UP".ALM_FLASHING, IsaTripFlashing := "UP".TRIP_FLASHING, Val_Out =>, Alm_Fail =>, Alm_HiHi =>, Alm_Hi =>, Alm_Lo =>, Alm_LoLo =>, Fo_Fail =>, Fo_HiHi =>, Fo_LoLo =>, SpareOut1 =>, SpareOut2 =>, SpareOut4 =>)
   END_RUNG
   // the same network as SCL:
   "PT_200B"(Inp_PV := "PT_200B_FLD",   // "SEID_AIn"
             Cfg_PVEUMin := "SETTINGS".PT_200.RANGE_H,
             Cfg_PVEUMax := "SETTINGS".PT_200.RANGE_L,
             Cfg_InpRawMin := 0,
             Cfg_InpRawMax := 27648,
             Cfg_FailRawHiLim := 29376,
             Cfg_FailRawLoLim := -691,
             Inp_PVBad := false,
             Cfg_FailBypass := false,
             Cfg_FailTripsUnit := true,
             Cfg_FailResetRequired := false,
             Cfg_InFailUsePVEUMax := "PT_200".Cfg_InFailUsePVEUMax,
             Cfg_InFailUsePVEUMin := "PT_200".Cfg_InFailUsePVEUMin,
             Cfg_InFailUseValSub := "PT_200".Cfg_InFailUseValSub,
             Cfg_ValSub := 0.0,
             Cfg_FailDelay := T#0ms,
             Cfg_HasHiHiAlm := "PT_200".Cfg_HasHiHiAlm,
             Oset_HiHiLim := "SETTINGS".PT_200.SP_HH,
             Cfg_HiHiDelay := T#1s,
             Cfg_HiHiDB := 0.0,
             Cfg_HiHiBypass := false,
             Cfg_HiHiTripsUnit := true,
             Cfg_HiHiResetRequired := false,
             Cfg_HasHiAlm := "PT_200".Cfg_HasHiAlm,
             Oset_HiLim := "SETTINGS".PT_200.SP_H,
             Cfg_HiDelay := T#1s,
             Cfg_HiDB := 0.0,
             Cfg_HiBypass := false,
             Cfg_HiResetRequired := false,
             Cfg_HasLoAlm := "PT_200".Cfg_HasLoAlm,
             Oset_LoLim := "SETTINGS".PT_200.SP_L,
             Cfg_LoDelay := T#1s,
             Cfg_LoDB := 0.0,
             Cfg_LoBypass := false,
             Cfg_LoResetRequired := false,
             Cfg_HasLoLoAlm := "PT_200".Cfg_HasLoLoAlm,
             Oset_LoLoLim := "SETTINGS".PT_200.SP_LL,
             Cfg_LoLoDelay := T#1s,
             Cfg_LoLoDB := 0.0,
             Cfg_LoLoBypass := false,
             Cfg_LoLoTripsUnit := false,
             Cfg_LoLoResetRequired := false,
             Inp_Reset := "RESET",
             PCmd_MOS := false,
             SpareIn1 := 0.0,
             SpareIn2 := 0.0,
             CommonFirstOut := "CMN_FO",
             IsaAlarmFlashing := "UP".ALM_FLASHING,
             IsaTripFlashing := "UP".TRIP_FLASHING);
END_REGION

REGION Network 9: AI 9
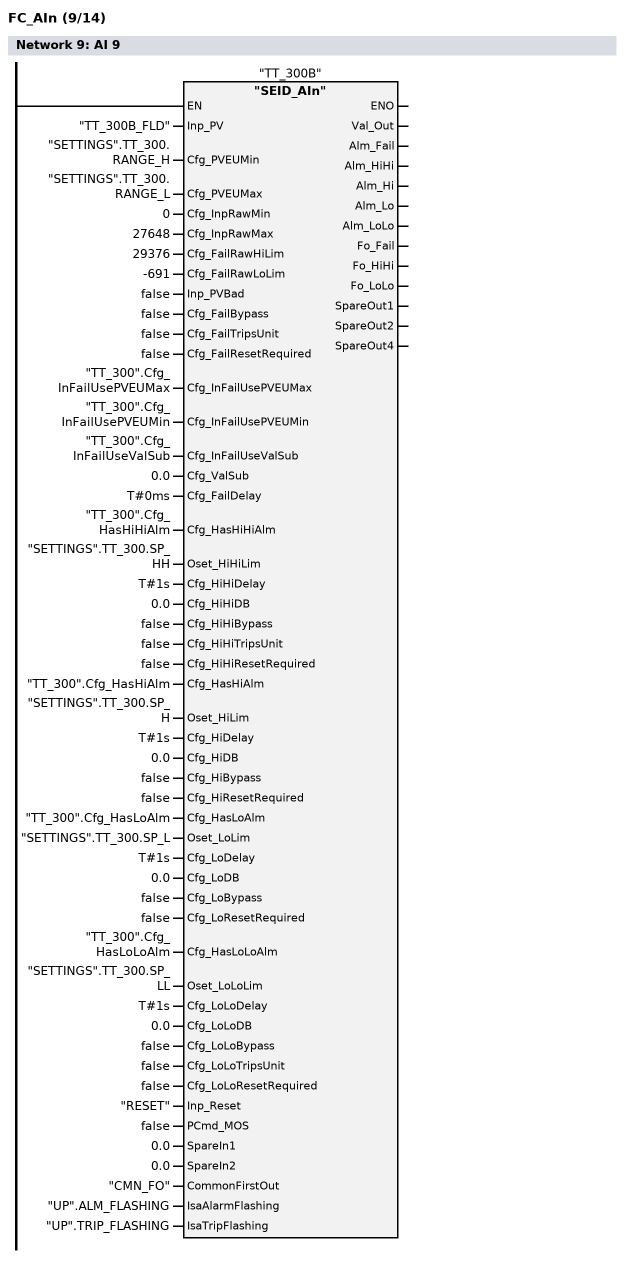
   RUNG wire#powerrail
      "TT_300B"(Inp_PV := "TT_300B_FLD", Cfg_PVEUMin := "SETTINGS".TT_300.RANGE_H, Cfg_PVEUMax := "SETTINGS".TT_300.RANGE_L, Cfg_InpRawMin := 0, Cfg_InpRawMax := 27648, Cfg_FailRawHiLim := 29376, Cfg_FailRawLoLim := -691, Inp_PVBad := false, Cfg_FailBypass := false, Cfg_FailTripsUnit := false, Cfg_FailResetRequired := false, Cfg_InFailUsePVEUMax := "TT_300".Cfg_InFailUsePVEUMax, Cfg_InFailUsePVEUMin := "TT_300".Cfg_InFailUsePVEUMin, Cfg_InFailUseValSub := "TT_300".Cfg_InFailUseValSub, Cfg_ValSub := 0.0, Cfg_FailDelay := T#0ms, Cfg_HasHiHiAlm := "TT_300".Cfg_HasHiHiAlm, Oset_HiHiLim := "SETTINGS".TT_300.SP_HH, Cfg_HiHiDelay := T#1s, Cfg_HiHiDB := 0.0, Cfg_HiHiBypass := false, Cfg_HiHiTripsUnit := false, Cfg_HiHiResetRequired := false, Cfg_HasHiAlm := "TT_300".Cfg_HasHiAlm, Oset_HiLim := "SETTINGS".TT_300.SP_H, Cfg_HiDelay := T#1s, Cfg_HiDB := 0.0, Cfg_HiBypass := false, Cfg_HiResetRequired := false, Cfg_HasLoAlm := "TT_300".Cfg_HasLoAlm, Oset_LoLim := "SETTINGS".TT_300.SP_L, Cfg_LoDelay := T#1s, Cfg_LoDB := 0.0, Cfg_LoBypass := false, Cfg_LoResetRequired := false, Cfg_HasLoLoAlm := "TT_300".Cfg_HasLoLoAlm, Oset_LoLoLim := "SETTINGS".TT_300.SP_LL, Cfg_LoLoDelay := T#1s, Cfg_LoLoDB := 0.0, Cfg_LoLoBypass := false, Cfg_LoLoTripsUnit := false, Cfg_LoLoResetRequired := false, Inp_Reset := "RESET", PCmd_MOS := false, SpareIn1 := 0.0, SpareIn2 := 0.0, CommonFirstOut := "CMN_FO", IsaAlarmFlashing := "UP".ALM_FLASHING, IsaTripFlashing := "UP".TRIP_FLASHING, Val_Out =>, Alm_Fail =>, Alm_HiHi =>, Alm_Hi =>, Alm_Lo =>, Alm_LoLo =>, Fo_Fail =>, Fo_HiHi =>, Fo_LoLo =>, SpareOut1 =>, SpareOut2 =>, SpareOut4 =>)
   END_RUNG
   // the same network as SCL:
   "TT_300B"(Inp_PV := "TT_300B_FLD",   // "SEID_AIn"
             Cfg_PVEUMin := "SETTINGS".TT_300.RANGE_H,
             Cfg_PVEUMax := "SETTINGS".TT_300.RANGE_L,
             Cfg_InpRawMin := 0,
             Cfg_InpRawMax := 27648,
             Cfg_FailRawHiLim := 29376,
             Cfg_FailRawLoLim := -691,
             Inp_PVBad := false,
             Cfg_FailBypass := false,
             Cfg_FailTripsUnit := false,
             Cfg_FailResetRequired := false,
             Cfg_InFailUsePVEUMax := "TT_300".Cfg_InFailUsePVEUMax,
             Cfg_InFailUsePVEUMin := "TT_300".Cfg_InFailUsePVEUMin,
             Cfg_InFailUseValSub := "TT_300".Cfg_InFailUseValSub,
             Cfg_ValSub := 0.0,
             Cfg_FailDelay := T#0ms,
             Cfg_HasHiHiAlm := "TT_300".Cfg_HasHiHiAlm,
             Oset_HiHiLim := "SETTINGS".TT_300.SP_HH,
             Cfg_HiHiDelay := T#1s,
             Cfg_HiHiDB := 0.0,
             Cfg_HiHiBypass := false,
             Cfg_HiHiTripsUnit := false,
             Cfg_HiHiResetRequired := false,
             Cfg_HasHiAlm := "TT_300".Cfg_HasHiAlm,
             Oset_HiLim := "SETTINGS".TT_300.SP_H,
             Cfg_HiDelay := T#1s,
             Cfg_HiDB := 0.0,
             Cfg_HiBypass := false,
             Cfg_HiResetRequired := false,
             Cfg_HasLoAlm := "TT_300".Cfg_HasLoAlm,
             Oset_LoLim := "SETTINGS".TT_300.SP_L,
             Cfg_LoDelay := T#1s,
             Cfg_LoDB := 0.0,
             Cfg_LoBypass := false,
             Cfg_LoResetRequired := false,
             Cfg_HasLoLoAlm := "TT_300".Cfg_HasLoLoAlm,
             Oset_LoLoLim := "SETTINGS".TT_300.SP_LL,
             Cfg_LoLoDelay := T#1s,
             Cfg_LoLoDB := 0.0,
             Cfg_LoLoBypass := false,
             Cfg_LoLoTripsUnit := false,
             Cfg_LoLoResetRequired := false,
             Inp_Reset := "RESET",
             PCmd_MOS := false,
             SpareIn1 := 0.0,
             SpareIn2 := 0.0,
             CommonFirstOut := "CMN_FO",
             IsaAlarmFlashing := "UP".ALM_FLASHING,
             IsaTripFlashing := "UP".TRIP_FLASHING);
END_REGION

REGION Network 10: AI 10
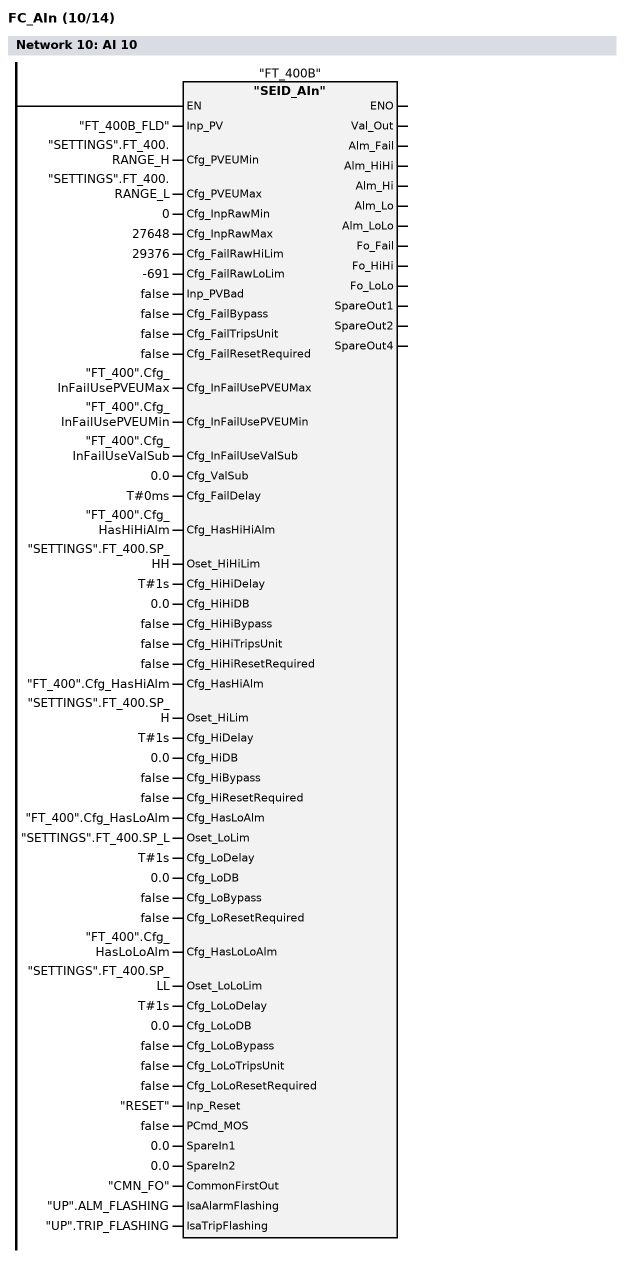
   RUNG wire#powerrail
      "FT_400B"(Inp_PV := "FT_400B_FLD", Cfg_PVEUMin := "SETTINGS".FT_400.RANGE_H, Cfg_PVEUMax := "SETTINGS".FT_400.RANGE_L, Cfg_InpRawMin := 0, Cfg_InpRawMax := 27648, Cfg_FailRawHiLim := 29376, Cfg_FailRawLoLim := -691, Inp_PVBad := false, Cfg_FailBypass := false, Cfg_FailTripsUnit := false, Cfg_FailResetRequired := false, Cfg_InFailUsePVEUMax := "FT_400".Cfg_InFailUsePVEUMax, Cfg_InFailUsePVEUMin := "FT_400".Cfg_InFailUsePVEUMin, Cfg_InFailUseValSub := "FT_400".Cfg_InFailUseValSub, Cfg_ValSub := 0.0, Cfg_FailDelay := T#0ms, Cfg_HasHiHiAlm := "FT_400".Cfg_HasHiHiAlm, Oset_HiHiLim := "SETTINGS".FT_400.SP_HH, Cfg_HiHiDelay := T#1s, Cfg_HiHiDB := 0.0, Cfg_HiHiBypass := false, Cfg_HiHiTripsUnit := false, Cfg_HiHiResetRequired := false, Cfg_HasHiAlm := "FT_400".Cfg_HasHiAlm, Oset_HiLim := "SETTINGS".FT_400.SP_H, Cfg_HiDelay := T#1s, Cfg_HiDB := 0.0, Cfg_HiBypass := false, Cfg_HiResetRequired := false, Cfg_HasLoAlm := "FT_400".Cfg_HasLoAlm, Oset_LoLim := "SETTINGS".FT_400.SP_L, Cfg_LoDelay := T#1s, Cfg_LoDB := 0.0, Cfg_LoBypass := false, Cfg_LoResetRequired := false, Cfg_HasLoLoAlm := "FT_400".Cfg_HasLoLoAlm, Oset_LoLoLim := "SETTINGS".FT_400.SP_LL, Cfg_LoLoDelay := T#1s, Cfg_LoLoDB := 0.0, Cfg_LoLoBypass := false, Cfg_LoLoTripsUnit := false, Cfg_LoLoResetRequired := false, Inp_Reset := "RESET", PCmd_MOS := false, SpareIn1 := 0.0, SpareIn2 := 0.0, CommonFirstOut := "CMN_FO", IsaAlarmFlashing := "UP".ALM_FLASHING, IsaTripFlashing := "UP".TRIP_FLASHING, Val_Out =>, Alm_Fail =>, Alm_HiHi =>, Alm_Hi =>, Alm_Lo =>, Alm_LoLo =>, Fo_Fail =>, Fo_HiHi =>, Fo_LoLo =>, SpareOut1 =>, SpareOut2 =>, SpareOut4 =>)
   END_RUNG
   // the same network as SCL:
   "FT_400B"(Inp_PV := "FT_400B_FLD",   // "SEID_AIn"
             Cfg_PVEUMin := "SETTINGS".FT_400.RANGE_H,
             Cfg_PVEUMax := "SETTINGS".FT_400.RANGE_L,
             Cfg_InpRawMin := 0,
             Cfg_InpRawMax := 27648,
             Cfg_FailRawHiLim := 29376,
             Cfg_FailRawLoLim := -691,
             Inp_PVBad := false,
             Cfg_FailBypass := false,
             Cfg_FailTripsUnit := false,
             Cfg_FailResetRequired := false,
             Cfg_InFailUsePVEUMax := "FT_400".Cfg_InFailUsePVEUMax,
             Cfg_InFailUsePVEUMin := "FT_400".Cfg_InFailUsePVEUMin,
             Cfg_InFailUseValSub := "FT_400".Cfg_InFailUseValSub,
             Cfg_ValSub := 0.0,
             Cfg_FailDelay := T#0ms,
             Cfg_HasHiHiAlm := "FT_400".Cfg_HasHiHiAlm,
             Oset_HiHiLim := "SETTINGS".FT_400.SP_HH,
             Cfg_HiHiDelay := T#1s,
             Cfg_HiHiDB := 0.0,
             Cfg_HiHiBypass := false,
             Cfg_HiHiTripsUnit := false,
             Cfg_HiHiResetRequired := false,
             Cfg_HasHiAlm := "FT_400".Cfg_HasHiAlm,
             Oset_HiLim := "SETTINGS".FT_400.SP_H,
             Cfg_HiDelay := T#1s,
             Cfg_HiDB := 0.0,
             Cfg_HiBypass := false,
             Cfg_HiResetRequired := false,
             Cfg_HasLoAlm := "FT_400".Cfg_HasLoAlm,
             Oset_LoLim := "SETTINGS".FT_400.SP_L,
             Cfg_LoDelay := T#1s,
             Cfg_LoDB := 0.0,
             Cfg_LoBypass := false,
             Cfg_LoResetRequired := false,
             Cfg_HasLoLoAlm := "FT_400".Cfg_HasLoLoAlm,
             Oset_LoLoLim := "SETTINGS".FT_400.SP_LL,
             Cfg_LoLoDelay := T#1s,
             Cfg_LoLoDB := 0.0,
             Cfg_LoLoBypass := false,
             Cfg_LoLoTripsUnit := false,
             Cfg_LoLoResetRequired := false,
             Inp_Reset := "RESET",
             PCmd_MOS := false,
             SpareIn1 := 0.0,
             SpareIn2 := 0.0,
             CommonFirstOut := "CMN_FO",
             IsaAlarmFlashing := "UP".ALM_FLASHING,
             IsaTripFlashing := "UP".TRIP_FLASHING);
END_REGION

REGION Network 11: AI 11
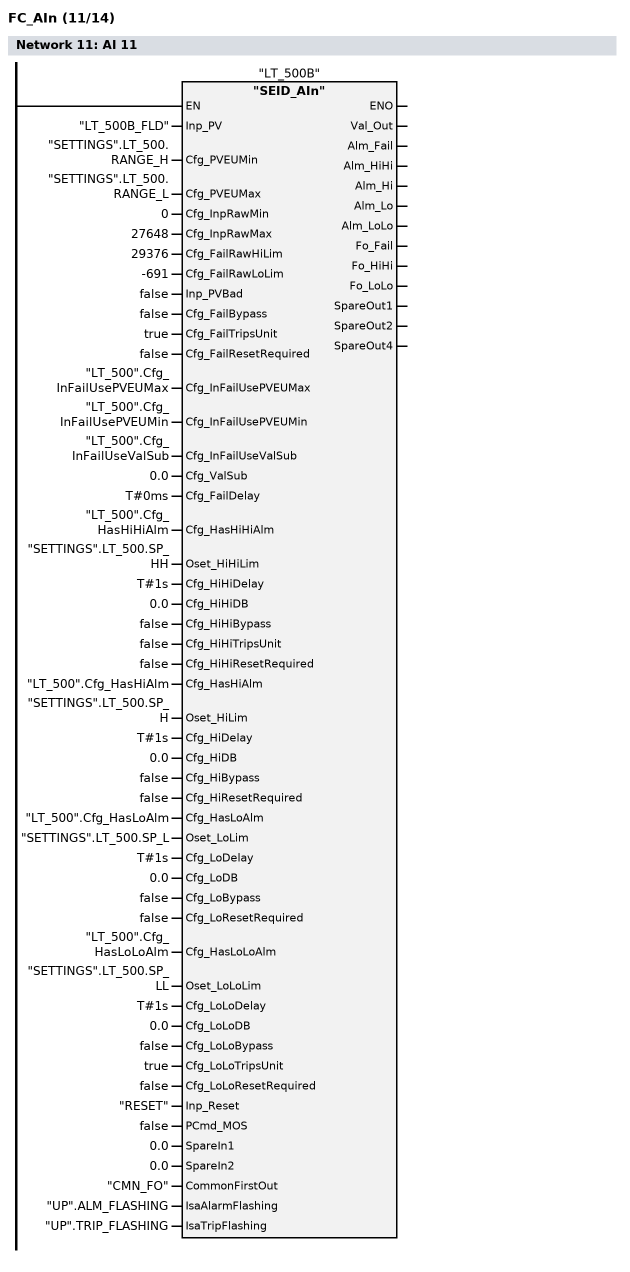
   RUNG wire#powerrail
      "LT_500B"(Inp_PV := "LT_500B_FLD", Cfg_PVEUMin := "SETTINGS".LT_500.RANGE_H, Cfg_PVEUMax := "SETTINGS".LT_500.RANGE_L, Cfg_InpRawMin := 0, Cfg_InpRawMax := 27648, Cfg_FailRawHiLim := 29376, Cfg_FailRawLoLim := -691, Inp_PVBad := false, Cfg_FailBypass := false, Cfg_FailTripsUnit := true, Cfg_FailResetRequired := false, Cfg_InFailUsePVEUMax := "LT_500".Cfg_InFailUsePVEUMax, Cfg_InFailUsePVEUMin := "LT_500".Cfg_InFailUsePVEUMin, Cfg_InFailUseValSub := "LT_500".Cfg_InFailUseValSub, Cfg_ValSub := 0.0, Cfg_FailDelay := T#0ms, Cfg_HasHiHiAlm := "LT_500".Cfg_HasHiHiAlm, Oset_HiHiLim := "SETTINGS".LT_500.SP_HH, Cfg_HiHiDelay := T#1s, Cfg_HiHiDB := 0.0, Cfg_HiHiBypass := false, Cfg_HiHiTripsUnit := false, Cfg_HiHiResetRequired := false, Cfg_HasHiAlm := "LT_500".Cfg_HasHiAlm, Oset_HiLim := "SETTINGS".LT_500.SP_H, Cfg_HiDelay := T#1s, Cfg_HiDB := 0.0, Cfg_HiBypass := false, Cfg_HiResetRequired := false, Cfg_HasLoAlm := "LT_500".Cfg_HasLoAlm, Oset_LoLim := "SETTINGS".LT_500.SP_L, Cfg_LoDelay := T#1s, Cfg_LoDB := 0.0, Cfg_LoBypass := false, Cfg_LoResetRequired := false, Cfg_HasLoLoAlm := "LT_500".Cfg_HasLoLoAlm, Oset_LoLoLim := "SETTINGS".LT_500.SP_LL, Cfg_LoLoDelay := T#1s, Cfg_LoLoDB := 0.0, Cfg_LoLoBypass := false, Cfg_LoLoTripsUnit := true, Cfg_LoLoResetRequired := false, Inp_Reset := "RESET", PCmd_MOS := false, SpareIn1 := 0.0, SpareIn2 := 0.0, CommonFirstOut := "CMN_FO", IsaAlarmFlashing := "UP".ALM_FLASHING, IsaTripFlashing := "UP".TRIP_FLASHING, Val_Out =>, Alm_Fail =>, Alm_HiHi =>, Alm_Hi =>, Alm_Lo =>, Alm_LoLo =>, Fo_Fail =>, Fo_HiHi =>, Fo_LoLo =>, SpareOut1 =>, SpareOut2 =>, SpareOut4 =>)
   END_RUNG
   // the same network as SCL:
   "LT_500B"(Inp_PV := "LT_500B_FLD",   // "SEID_AIn"
             Cfg_PVEUMin := "SETTINGS".LT_500.RANGE_H,
             Cfg_PVEUMax := "SETTINGS".LT_500.RANGE_L,
             Cfg_InpRawMin := 0,
             Cfg_InpRawMax := 27648,
             Cfg_FailRawHiLim := 29376,
             Cfg_FailRawLoLim := -691,
             Inp_PVBad := false,
             Cfg_FailBypass := false,
             Cfg_FailTripsUnit := true,
             Cfg_FailResetRequired := false,
             Cfg_InFailUsePVEUMax := "LT_500".Cfg_InFailUsePVEUMax,
             Cfg_InFailUsePVEUMin := "LT_500".Cfg_InFailUsePVEUMin,
             Cfg_InFailUseValSub := "LT_500".Cfg_InFailUseValSub,
             Cfg_ValSub := 0.0,
             Cfg_FailDelay := T#0ms,
             Cfg_HasHiHiAlm := "LT_500".Cfg_HasHiHiAlm,
             Oset_HiHiLim := "SETTINGS".LT_500.SP_HH,
             Cfg_HiHiDelay := T#1s,
             Cfg_HiHiDB := 0.0,
             Cfg_HiHiBypass := false,
             Cfg_HiHiTripsUnit := false,
             Cfg_HiHiResetRequired := false,
             Cfg_HasHiAlm := "LT_500".Cfg_HasHiAlm,
             Oset_HiLim := "SETTINGS".LT_500.SP_H,
             Cfg_HiDelay := T#1s,
             Cfg_HiDB := 0.0,
             Cfg_HiBypass := false,
             Cfg_HiResetRequired := false,
             Cfg_HasLoAlm := "LT_500".Cfg_HasLoAlm,
             Oset_LoLim := "SETTINGS".LT_500.SP_L,
             Cfg_LoDelay := T#1s,
             Cfg_LoDB := 0.0,
             Cfg_LoBypass := false,
             Cfg_LoResetRequired := false,
             Cfg_HasLoLoAlm := "LT_500".Cfg_HasLoLoAlm,
             Oset_LoLoLim := "SETTINGS".LT_500.SP_LL,
             Cfg_LoLoDelay := T#1s,
             Cfg_LoLoDB := 0.0,
             Cfg_LoLoBypass := false,
             Cfg_LoLoTripsUnit := true,
             Cfg_LoLoResetRequired := false,
             Inp_Reset := "RESET",
             PCmd_MOS := false,
             SpareIn1 := 0.0,
             SpareIn2 := 0.0,
             CommonFirstOut := "CMN_FO",
             IsaAlarmFlashing := "UP".ALM_FLASHING,
             IsaTripFlashing := "UP".TRIP_FLASHING);
END_REGION

REGION Network 12: AI 12
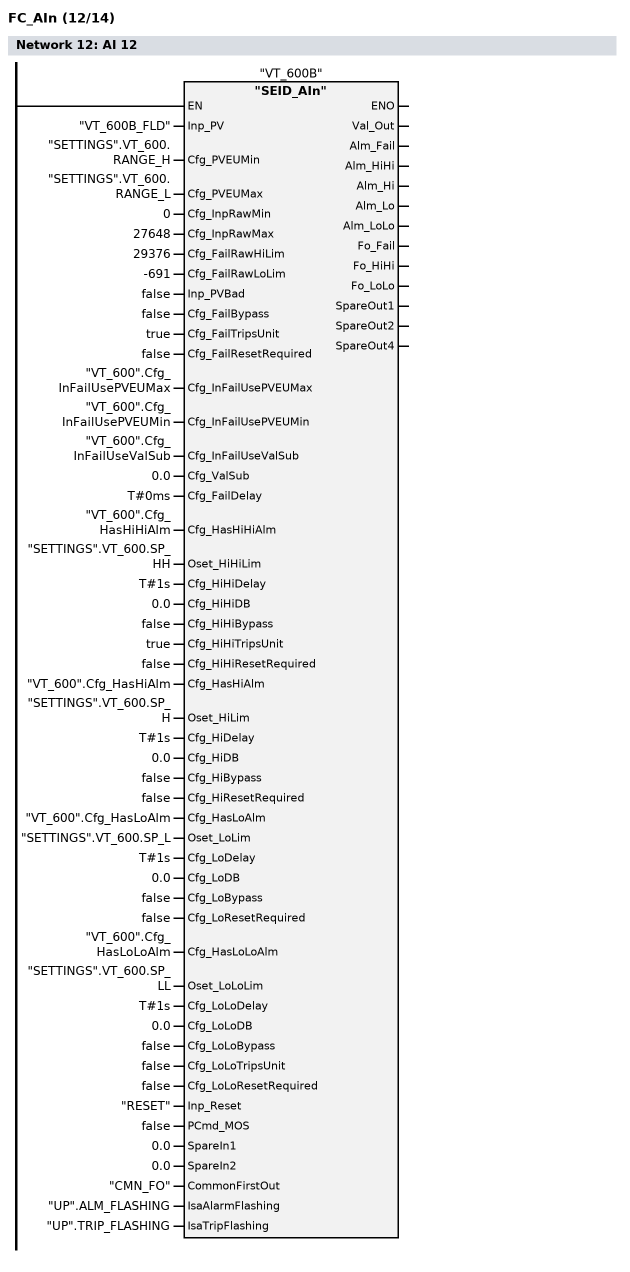
   RUNG wire#powerrail
      "VT_600B"(Inp_PV := "VT_600B_FLD", Cfg_PVEUMin := "SETTINGS".VT_600.RANGE_H, Cfg_PVEUMax := "SETTINGS".VT_600.RANGE_L, Cfg_InpRawMin := 0, Cfg_InpRawMax := 27648, Cfg_FailRawHiLim := 29376, Cfg_FailRawLoLim := -691, Inp_PVBad := false, Cfg_FailBypass := false, Cfg_FailTripsUnit := true, Cfg_FailResetRequired := false, Cfg_InFailUsePVEUMax := "VT_600".Cfg_InFailUsePVEUMax, Cfg_InFailUsePVEUMin := "VT_600".Cfg_InFailUsePVEUMin, Cfg_InFailUseValSub := "VT_600".Cfg_InFailUseValSub, Cfg_ValSub := 0.0, Cfg_FailDelay := T#0ms, Cfg_HasHiHiAlm := "VT_600".Cfg_HasHiHiAlm, Oset_HiHiLim := "SETTINGS".VT_600.SP_HH, Cfg_HiHiDelay := T#1s, Cfg_HiHiDB := 0.0, Cfg_HiHiBypass := false, Cfg_HiHiTripsUnit := true, Cfg_HiHiResetRequired := false, Cfg_HasHiAlm := "VT_600".Cfg_HasHiAlm, Oset_HiLim := "SETTINGS".VT_600.SP_H, Cfg_HiDelay := T#1s, Cfg_HiDB := 0.0, Cfg_HiBypass := false, Cfg_HiResetRequired := false, Cfg_HasLoAlm := "VT_600".Cfg_HasLoAlm, Oset_LoLim := "SETTINGS".VT_600.SP_L, Cfg_LoDelay := T#1s, Cfg_LoDB := 0.0, Cfg_LoBypass := false, Cfg_LoResetRequired := false, Cfg_HasLoLoAlm := "VT_600".Cfg_HasLoLoAlm, Oset_LoLoLim := "SETTINGS".VT_600.SP_LL, Cfg_LoLoDelay := T#1s, Cfg_LoLoDB := 0.0, Cfg_LoLoBypass := false, Cfg_LoLoTripsUnit := false, Cfg_LoLoResetRequired := false, Inp_Reset := "RESET", PCmd_MOS := false, SpareIn1 := 0.0, SpareIn2 := 0.0, CommonFirstOut := "CMN_FO", IsaAlarmFlashing := "UP".ALM_FLASHING, IsaTripFlashing := "UP".TRIP_FLASHING, Val_Out =>, Alm_Fail =>, Alm_HiHi =>, Alm_Hi =>, Alm_Lo =>, Alm_LoLo =>, Fo_Fail =>, Fo_HiHi =>, Fo_LoLo =>, SpareOut1 =>, SpareOut2 =>, SpareOut4 =>)
   END_RUNG
   // the same network as SCL:
   "VT_600B"(Inp_PV := "VT_600B_FLD",   // "SEID_AIn"
             Cfg_PVEUMin := "SETTINGS".VT_600.RANGE_H,
             Cfg_PVEUMax := "SETTINGS".VT_600.RANGE_L,
             Cfg_InpRawMin := 0,
             Cfg_InpRawMax := 27648,
             Cfg_FailRawHiLim := 29376,
             Cfg_FailRawLoLim := -691,
             Inp_PVBad := false,
             Cfg_FailBypass := false,
             Cfg_FailTripsUnit := true,
             Cfg_FailResetRequired := false,
             Cfg_InFailUsePVEUMax := "VT_600".Cfg_InFailUsePVEUMax,
             Cfg_InFailUsePVEUMin := "VT_600".Cfg_InFailUsePVEUMin,
             Cfg_InFailUseValSub := "VT_600".Cfg_InFailUseValSub,
             Cfg_ValSub := 0.0,
             Cfg_FailDelay := T#0ms,
             Cfg_HasHiHiAlm := "VT_600".Cfg_HasHiHiAlm,
             Oset_HiHiLim := "SETTINGS".VT_600.SP_HH,
             Cfg_HiHiDelay := T#1s,
             Cfg_HiHiDB := 0.0,
             Cfg_HiHiBypass := false,
             Cfg_HiHiTripsUnit := true,
             Cfg_HiHiResetRequired := false,
             Cfg_HasHiAlm := "VT_600".Cfg_HasHiAlm,
             Oset_HiLim := "SETTINGS".VT_600.SP_H,
             Cfg_HiDelay := T#1s,
             Cfg_HiDB := 0.0,
             Cfg_HiBypass := false,
             Cfg_HiResetRequired := false,
             Cfg_HasLoAlm := "VT_600".Cfg_HasLoAlm,
             Oset_LoLim := "SETTINGS".VT_600.SP_L,
             Cfg_LoDelay := T#1s,
             Cfg_LoDB := 0.0,
             Cfg_LoBypass := false,
             Cfg_LoResetRequired := false,
             Cfg_HasLoLoAlm := "VT_600".Cfg_HasLoLoAlm,
             Oset_LoLoLim := "SETTINGS".VT_600.SP_LL,
             Cfg_LoLoDelay := T#1s,
             Cfg_LoLoDB := 0.0,
             Cfg_LoLoBypass := false,
             Cfg_LoLoTripsUnit := false,
             Cfg_LoLoResetRequired := false,
             Inp_Reset := "RESET",
             PCmd_MOS := false,
             SpareIn1 := 0.0,
             SpareIn2 := 0.0,
             CommonFirstOut := "CMN_FO",
             IsaAlarmFlashing := "UP".ALM_FLASHING,
             IsaTripFlashing := "UP".TRIP_FLASHING);
END_REGION

REGION Network 13: AI 13
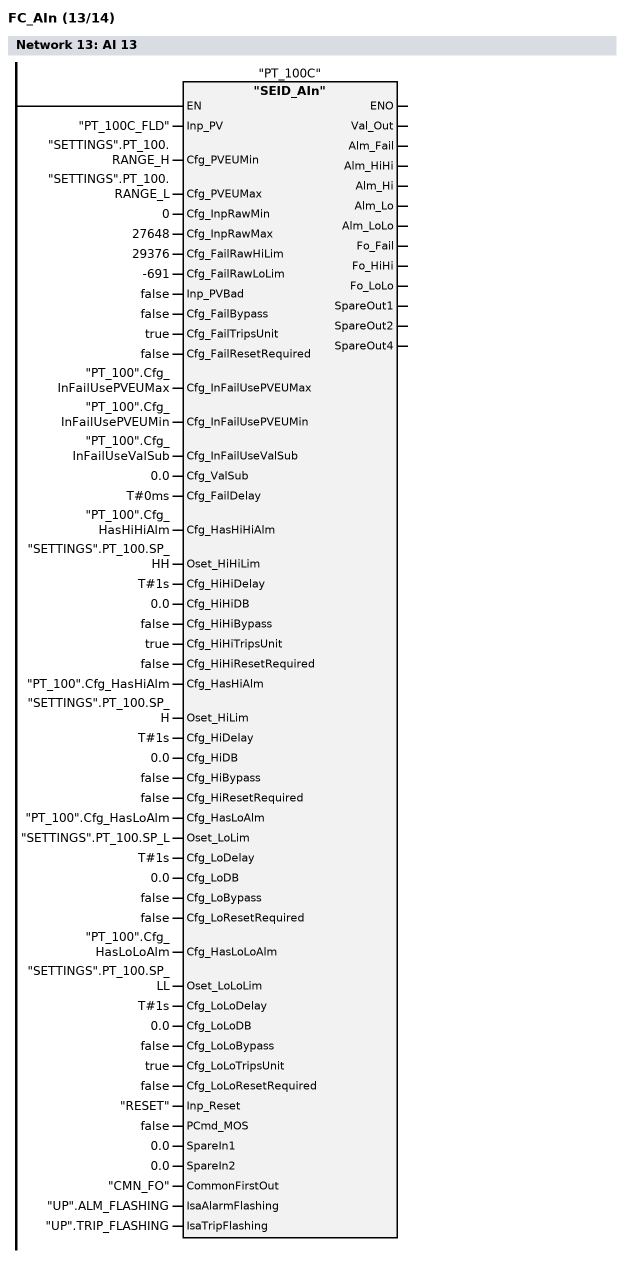
   RUNG wire#powerrail
      "PT_100C"(Inp_PV := "PT_100C_FLD", Cfg_PVEUMin := "SETTINGS".PT_100.RANGE_H, Cfg_PVEUMax := "SETTINGS".PT_100.RANGE_L, Cfg_InpRawMin := 0, Cfg_InpRawMax := 27648, Cfg_FailRawHiLim := 29376, Cfg_FailRawLoLim := -691, Inp_PVBad := false, Cfg_FailBypass := false, Cfg_FailTripsUnit := true, Cfg_FailResetRequired := false, Cfg_InFailUsePVEUMax := "PT_100".Cfg_InFailUsePVEUMax, Cfg_InFailUsePVEUMin := "PT_100".Cfg_InFailUsePVEUMin, Cfg_InFailUseValSub := "PT_100".Cfg_InFailUseValSub, Cfg_ValSub := 0.0, Cfg_FailDelay := T#0ms, Cfg_HasHiHiAlm := "PT_100".Cfg_HasHiHiAlm, Oset_HiHiLim := "SETTINGS".PT_100.SP_HH, Cfg_HiHiDelay := T#1s, Cfg_HiHiDB := 0.0, Cfg_HiHiBypass := false, Cfg_HiHiTripsUnit := true, Cfg_HiHiResetRequired := false, Cfg_HasHiAlm := "PT_100".Cfg_HasHiAlm, Oset_HiLim := "SETTINGS".PT_100.SP_H, Cfg_HiDelay := T#1s, Cfg_HiDB := 0.0, Cfg_HiBypass := false, Cfg_HiResetRequired := false, Cfg_HasLoAlm := "PT_100".Cfg_HasLoAlm, Oset_LoLim := "SETTINGS".PT_100.SP_L, Cfg_LoDelay := T#1s, Cfg_LoDB := 0.0, Cfg_LoBypass := false, Cfg_LoResetRequired := false, Cfg_HasLoLoAlm := "PT_100".Cfg_HasLoLoAlm, Oset_LoLoLim := "SETTINGS".PT_100.SP_LL, Cfg_LoLoDelay := T#1s, Cfg_LoLoDB := 0.0, Cfg_LoLoBypass := false, Cfg_LoLoTripsUnit := true, Cfg_LoLoResetRequired := false, Inp_Reset := "RESET", PCmd_MOS := false, SpareIn1 := 0.0, SpareIn2 := 0.0, CommonFirstOut := "CMN_FO", IsaAlarmFlashing := "UP".ALM_FLASHING, IsaTripFlashing := "UP".TRIP_FLASHING, Val_Out =>, Alm_Fail =>, Alm_HiHi =>, Alm_Hi =>, Alm_Lo =>, Alm_LoLo =>, Fo_Fail =>, Fo_HiHi =>, Fo_LoLo =>, SpareOut1 =>, SpareOut2 =>, SpareOut4 =>)
   END_RUNG
   // the same network as SCL:
   "PT_100C"(Inp_PV := "PT_100C_FLD",   // "SEID_AIn"
             Cfg_PVEUMin := "SETTINGS".PT_100.RANGE_H,
             Cfg_PVEUMax := "SETTINGS".PT_100.RANGE_L,
             Cfg_InpRawMin := 0,
             Cfg_InpRawMax := 27648,
             Cfg_FailRawHiLim := 29376,
             Cfg_FailRawLoLim := -691,
             Inp_PVBad := false,
             Cfg_FailBypass := false,
             Cfg_FailTripsUnit := true,
             Cfg_FailResetRequired := false,
             Cfg_InFailUsePVEUMax := "PT_100".Cfg_InFailUsePVEUMax,
             Cfg_InFailUsePVEUMin := "PT_100".Cfg_InFailUsePVEUMin,
             Cfg_InFailUseValSub := "PT_100".Cfg_InFailUseValSub,
             Cfg_ValSub := 0.0,
             Cfg_FailDelay := T#0ms,
             Cfg_HasHiHiAlm := "PT_100".Cfg_HasHiHiAlm,
             Oset_HiHiLim := "SETTINGS".PT_100.SP_HH,
             Cfg_HiHiDelay := T#1s,
             Cfg_HiHiDB := 0.0,
             Cfg_HiHiBypass := false,
             Cfg_HiHiTripsUnit := true,
             Cfg_HiHiResetRequired := false,
             Cfg_HasHiAlm := "PT_100".Cfg_HasHiAlm,
             Oset_HiLim := "SETTINGS".PT_100.SP_H,
             Cfg_HiDelay := T#1s,
             Cfg_HiDB := 0.0,
             Cfg_HiBypass := false,
             Cfg_HiResetRequired := false,
             Cfg_HasLoAlm := "PT_100".Cfg_HasLoAlm,
             Oset_LoLim := "SETTINGS".PT_100.SP_L,
             Cfg_LoDelay := T#1s,
             Cfg_LoDB := 0.0,
             Cfg_LoBypass := false,
             Cfg_LoResetRequired := false,
             Cfg_HasLoLoAlm := "PT_100".Cfg_HasLoLoAlm,
             Oset_LoLoLim := "SETTINGS".PT_100.SP_LL,
             Cfg_LoLoDelay := T#1s,
             Cfg_LoLoDB := 0.0,
             Cfg_LoLoBypass := false,
             Cfg_LoLoTripsUnit := true,
             Cfg_LoLoResetRequired := false,
             Inp_Reset := "RESET",
             PCmd_MOS := false,
             SpareIn1 := 0.0,
             SpareIn2 := 0.0,
             CommonFirstOut := "CMN_FO",
             IsaAlarmFlashing := "UP".ALM_FLASHING,
             IsaTripFlashing := "UP".TRIP_FLASHING);
END_REGION

REGION Network 14: AI 14
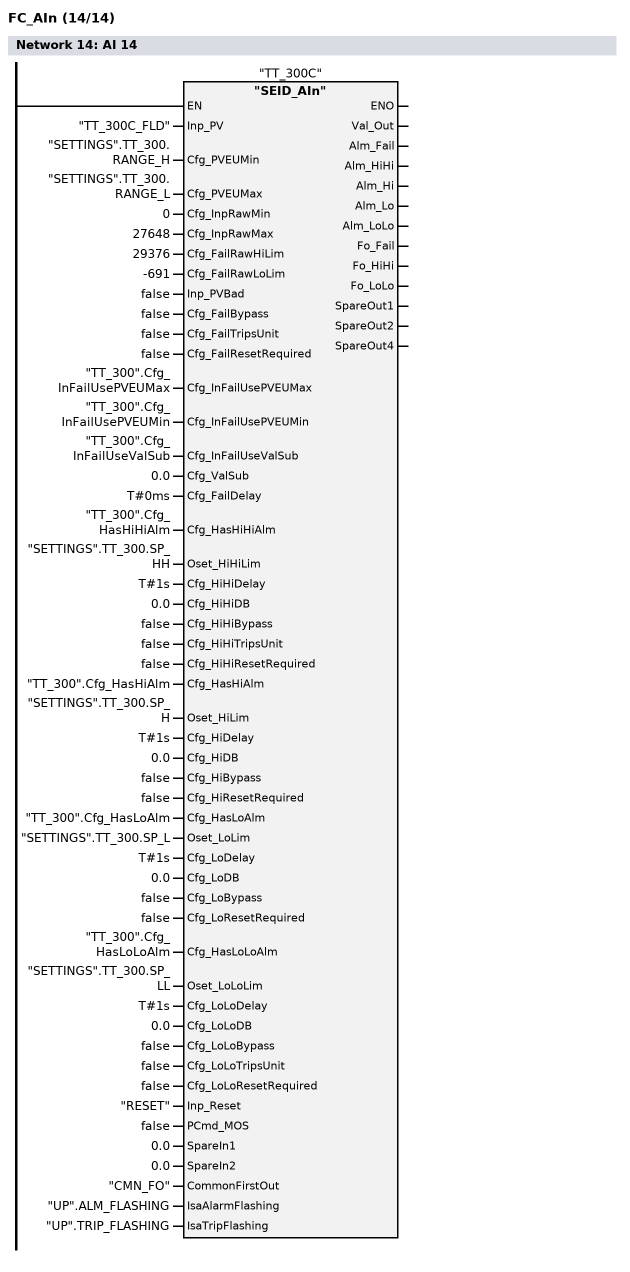
   RUNG wire#powerrail
      "TT_300C"(Inp_PV := "TT_300C_FLD", Cfg_PVEUMin := "SETTINGS".TT_300.RANGE_H, Cfg_PVEUMax := "SETTINGS".TT_300.RANGE_L, Cfg_InpRawMin := 0, Cfg_InpRawMax := 27648, Cfg_FailRawHiLim := 29376, Cfg_FailRawLoLim := -691, Inp_PVBad := false, Cfg_FailBypass := false, Cfg_FailTripsUnit := false, Cfg_FailResetRequired := false, Cfg_InFailUsePVEUMax := "TT_300".Cfg_InFailUsePVEUMax, Cfg_InFailUsePVEUMin := "TT_300".Cfg_InFailUsePVEUMin, Cfg_InFailUseValSub := "TT_300".Cfg_InFailUseValSub, Cfg_ValSub := 0.0, Cfg_FailDelay := T#0ms, Cfg_HasHiHiAlm := "TT_300".Cfg_HasHiHiAlm, Oset_HiHiLim := "SETTINGS".TT_300.SP_HH, Cfg_HiHiDelay := T#1s, Cfg_HiHiDB := 0.0, Cfg_HiHiBypass := false, Cfg_HiHiTripsUnit := false, Cfg_HiHiResetRequired := false, Cfg_HasHiAlm := "TT_300".Cfg_HasHiAlm, Oset_HiLim := "SETTINGS".TT_300.SP_H, Cfg_HiDelay := T#1s, Cfg_HiDB := 0.0, Cfg_HiBypass := false, Cfg_HiResetRequired := false, Cfg_HasLoAlm := "TT_300".Cfg_HasLoAlm, Oset_LoLim := "SETTINGS".TT_300.SP_L, Cfg_LoDelay := T#1s, Cfg_LoDB := 0.0, Cfg_LoBypass := false, Cfg_LoResetRequired := false, Cfg_HasLoLoAlm := "TT_300".Cfg_HasLoLoAlm, Oset_LoLoLim := "SETTINGS".TT_300.SP_LL, Cfg_LoLoDelay := T#1s, Cfg_LoLoDB := 0.0, Cfg_LoLoBypass := false, Cfg_LoLoTripsUnit := false, Cfg_LoLoResetRequired := false, Inp_Reset := "RESET", PCmd_MOS := false, SpareIn1 := 0.0, SpareIn2 := 0.0, CommonFirstOut := "CMN_FO", IsaAlarmFlashing := "UP".ALM_FLASHING, IsaTripFlashing := "UP".TRIP_FLASHING, Val_Out =>, Alm_Fail =>, Alm_HiHi =>, Alm_Hi =>, Alm_Lo =>, Alm_LoLo =>, Fo_Fail =>, Fo_HiHi =>, Fo_LoLo =>, SpareOut1 =>, SpareOut2 =>, SpareOut4 =>)
   END_RUNG
   // the same network as SCL:
   "TT_300C"(Inp_PV := "TT_300C_FLD",   // "SEID_AIn"
             Cfg_PVEUMin := "SETTINGS".TT_300.RANGE_H,
             Cfg_PVEUMax := "SETTINGS".TT_300.RANGE_L,
             Cfg_InpRawMin := 0,
             Cfg_InpRawMax := 27648,
             Cfg_FailRawHiLim := 29376,
             Cfg_FailRawLoLim := -691,
             Inp_PVBad := false,
             Cfg_FailBypass := false,
             Cfg_FailTripsUnit := false,
             Cfg_FailResetRequired := false,
             Cfg_InFailUsePVEUMax := "TT_300".Cfg_InFailUsePVEUMax,
             Cfg_InFailUsePVEUMin := "TT_300".Cfg_InFailUsePVEUMin,
             Cfg_InFailUseValSub := "TT_300".Cfg_InFailUseValSub,
             Cfg_ValSub := 0.0,
             Cfg_FailDelay := T#0ms,
             Cfg_HasHiHiAlm := "TT_300".Cfg_HasHiHiAlm,
             Oset_HiHiLim := "SETTINGS".TT_300.SP_HH,
             Cfg_HiHiDelay := T#1s,
             Cfg_HiHiDB := 0.0,
             Cfg_HiHiBypass := false,
             Cfg_HiHiTripsUnit := false,
             Cfg_HiHiResetRequired := false,
             Cfg_HasHiAlm := "TT_300".Cfg_HasHiAlm,
             Oset_HiLim := "SETTINGS".TT_300.SP_H,
             Cfg_HiDelay := T#1s,
             Cfg_HiDB := 0.0,
             Cfg_HiBypass := false,
             Cfg_HiResetRequired := false,
             Cfg_HasLoAlm := "TT_300".Cfg_HasLoAlm,
             Oset_LoLim := "SETTINGS".TT_300.SP_L,
             Cfg_LoDelay := T#1s,
             Cfg_LoDB := 0.0,
             Cfg_LoBypass := false,
             Cfg_LoResetRequired := false,
             Cfg_HasLoLoAlm := "TT_300".Cfg_HasLoLoAlm,
             Oset_LoLoLim := "SETTINGS".TT_300.SP_LL,
             Cfg_LoLoDelay := T#1s,
             Cfg_LoLoDB := 0.0,
             Cfg_LoLoBypass := false,
             Cfg_LoLoTripsUnit := false,
             Cfg_LoLoResetRequired := false,
             Inp_Reset := "RESET",
             PCmd_MOS := false,
             SpareIn1 := 0.0,
             SpareIn2 := 0.0,
             CommonFirstOut := "CMN_FO",
             IsaAlarmFlashing := "UP".ALM_FLASHING,
             IsaTripFlashing := "UP".TRIP_FLASHING);
END_REGION
END_FUNCTION
